KUKA KRL program: EPS_2_25694_CR03_A_20260114065856.src

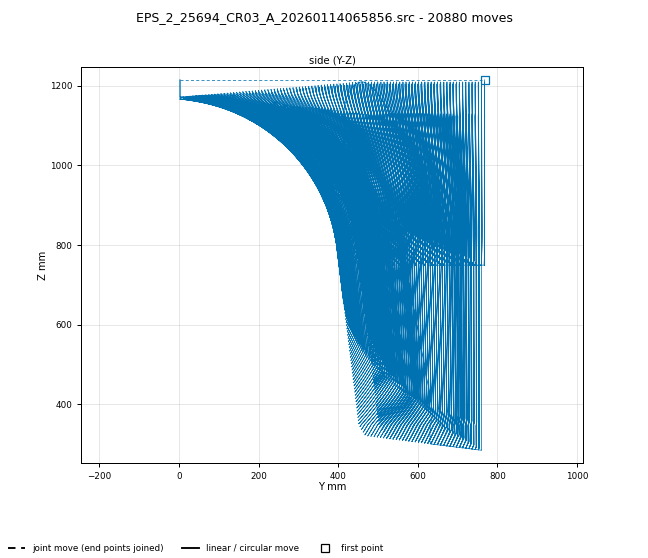
[picture p0: tool path of EPS_2_25694_CR03_A_20260114065856.src, 20880 of 20882 moves have a stored position in this frame; points joined in program order, loops and branches not executed]
&ACCESS RVP
&REL 4
&COMMENT QRS 19112012
&PARAM EDITMASK = *
DEF PART()
EXT BAS (BAS_COMMAND :IN,REAL :IN )
INT I
BAS (#INITMOV,0 )

;KUKA QRS Post kuka4.cps  Date:22-06-2017 !

File_ID=2973

QRS_PRE_INIT()

;Init var - Until changes are made in qrs_pre_init
Outlet_Square_prg=0
Inlet_1_Square_prg=0
Inlet_2_Square_prg=0
Inlet_3_Square_prg=0
Inlet_4_Square_prg=0
Inlet_5_Square_prg=0

Outlet_1={X 0.000, Y 457.000, Z 786.000, B 0.000, E1 0.000 }
Inlet_1={X 0.000, Y 514.000, Z 744.000, B 0.000, E1 189.000 }
Outlet_1_type=838
Inlet_1_type=762
;QRS#1=Sidecore dimensions
;QRS#2=825-33" Concrete
;QRS#3=750-30" Concrete
;QRS#4=
;QRS#5=
;QRS#6=
;QRS#7=
;QRS#8=
;QRS#9=S306-46
;QRS#10=S306-42L
;QRS#11=
;QRS#12=
;QRS#13=
;QRS#14=
;QRS#15=
;QRS#16=1524x152x1676 5,5'
;QRS#17=EPS Height
;QRS#18=1205
;QRS#19=*
;QRS#20= UPDATED VERSION 22-06-2017
;QRS#21=*
Outlet_Square=0650
Inlet_1_Square=0550
Inlet_2_Square=0
Inlet_3_Square=0
Inlet_4_Square=0
Inlet_5_Square=0
Mill_Square=1
Outlet_Square_Prg=267
Inlet_1_Square_prg=266

QRS_INIT()

$ADVANCE=5

; T1
PTP {E1 173.009,E2 173.009}
PTP {X 0,Y 767.725,A -85,B 0,C 180,E1 173.009,E2 173.009,E3 0,E4 0,E5 0,E6 0}
QRS_SPEED_INIT()
LIN {X 0,Y 767.725,Z 1215,A -85,B 0,C 180,E1 173.009,E2 173.009,E3 0,E4 0,E5 0,E6 0} C_VEL
LIN {X 0,Y 767.725,Z 751.56,A -85,B 0,C 180,E1 173.009,E2 173.009} C_VEL
LIN {X 0,Y 767.762,Z 749.56,A -85,B 0,C 180,E1 173.158,E2 173.158} C_VEL
LIN {X 0,Y 767.852,Z 749.56,A -85,B 0,C 180,E1 173.458,E2 173.458} C_VEL
LIN {X 0,Y 767.871,Z 749.56,A -85,B 0,C 180,E1 177.201,E2 177.201} C_VEL
LIN {X 0,Y 767.875,Z 749.56,A -85,B 0,C 180,E1 180.933,E2 180.933} C_VEL
LIN {X 0,Y 767.854,Z 749.56,A -85,B 0,C 180,E1 184.668,E2 184.668} C_VEL
LIN {X 0,Y 767.837,Z 749.56,A -85,B 0,C 180,E1 188.423,E2 188.423} C_VEL
LIN {X 0,Y 767.811,Z 749.56,A -85,B 0,C 180,E1 192.216,E2 192.216} C_VEL
LIN {X 0,Y 767.861,Z 749.56,A -85,B 0,C 180,E1 196.219,E2 196.219} C_VEL
LIN {X 0,Y 767.815,Z 749.56,A -85,B 0,C 180,E1 199.987,E2 199.987} C_VEL
LIN {X 0,Y 767.797,Z 749.56,A -85,B 0,C 180,E1 204.011,E2 204.011} C_VEL
LIN {X 0,Y 767.777,Z 749.56,A -85,B 0,C 180,E1 208.166,E2 208.166} C_VEL
LIN {X 0,Y 767.322,Z 749.56,A -85,B 0,C 180,E1 210.327,E2 210.327} C_VEL
LIN {X 0,Y 767.741,Z 749.56,A -85,B 0,C 180,E1 212.491,E2 212.491} C_VEL
LIN {X 0,Y 767.429,Z 749.56,A -85,B 0,C 180,E1 213.853,E2 213.853} C_VEL
LIN {X 0,Y 767.751,Z 749.56,A -85,B 0,C 180,E1 217.101,E2 217.101} C_VEL
LIN {X 0,Y 767.178,Z 749.56,A -85,B 0,C 180,E1 220.041,E2 220.041} C_VEL
LIN {X 0,Y 767.652,Z 749.56,A -85,B 0,C 180,E1 221.872,E2 221.872} C_VEL
LIN {X 0,Y 767.68,Z 749.56,A -85,B 0,C 180,E1 222.901,E2 222.901} C_VEL
LIN {X 0,Y 767.683,Z 749.56,A -85,B 0,C 180,E1 224.427,E2 224.427} C_VEL
LIN {X 0,Y 767.65,Z 749.56,A -85,B 0,C 180,E1 225.573,E2 225.573} C_VEL
LIN {X 0,Y 767.7,Z 749.56,A -85,B 0,C 180,E1 229.915,E2 229.915} C_VEL
LIN {X 0,Y 767.764,Z 749.56,A -85,B 0,C 180,E1 230.596,E2 230.596} C_VEL
LIN {X 0,Y 767.72,Z 749.56,A -85,B 0,C 180,E1 232.967,E2 232.967} C_VEL
LIN {X 0,Y 767.714,Z 749.56,A -85,B 0,C 180,E1 233.556,E2 233.556} C_VEL
LIN {X 0,Y 766.586,Z 750.428,A -85,B 0,C 180,E1 233.715,E2 233.715} C_VEL
LIN {X 0,Y 767.117,Z 773.995,A -85,B 0,C 180,E1 234.011,E2 234.011} C_VEL
LIN {X 0,Y 767.163,Z 809.122,A -85,B 0,C 180,E1 234.411,E2 234.411} C_VEL
LIN {X 0,Y 767.457,Z 829.921,A -85,B 0,C 180,E1 234.684,E2 234.684} C_VEL
LIN {X 0,Y 767.407,Z 846.164,A -85,B 0,C 180,E1 234.938,E2 234.938} C_VEL
LIN {X 0,Y 767.21,Z 858.585,A -85,B 0,C 180,E1 235.165,E2 235.165} C_VEL
LIN {X 0,Y 767.328,Z 875.217,A -85,B 0,C 180,E1 235.536,E2 235.536} C_VEL
LIN {X 0,Y 767.282,Z 887.767,A -85,B 0,C 180,E1 235.85,E2 235.85} C_VEL
LIN {X 0,Y 767.451,Z 900.804,A -85,B 0,C 180,E1 236.23,E2 236.23} C_VEL
LIN {X 0,Y 767.479,Z 917.969,A -85,B 0,C 180,E1 236.766,E2 236.766} C_VEL
LIN {X 0,Y 767.395,Z 931.208,A -85,B 0,C 180,E1 237.225,E2 237.225} C_VEL
LIN {X 0,Y 767.51,Z 940.173,A -85,B 0,C 180,E1 237.569,E2 237.569} C_VEL
LIN {X 0,Y 767.582,Z 955.64,A -85,B 0,C 180,E1 238.192,E2 238.192} C_VEL
LIN {X 0,Y 767.448,Z 974.022,A -85,B 0,C 180,E1 239.005,E2 239.005} C_VEL
LIN {X 0,Y 767.587,Z 991.208,A -85,B 0,C 180,E1 239.856,E2 239.856} C_VEL
LIN {X 0,Y 767.619,Z 1008.156,A -85,B 0,C 180,E1 240.771,E2 240.771} C_VEL
LIN {X 0,Y 767.612,Z 1024.962,A -85,B 0,C 180,E1 241.762,E2 241.762} C_VEL
LIN {X 0,Y 767.627,Z 1040.383,A -85,B 0,C 180,E1 242.751,E2 242.751} C_VEL
LIN {X 0,Y 767.65,Z 1055.737,A -85,B 0,C 180,E1 243.819,E2 243.819} C_VEL
LIN {X 0,Y 767.579,Z 1070.87,A -85,B 0,C 180,E1 244.96,E2 244.96} C_VEL
LIN {X 0,Y 767.603,Z 1083.468,A -85,B 0,C 180,E1 245.983,E2 245.983} C_VEL
LIN {X 0,Y 767.694,Z 1096.523,A -85,B 0,C 180,E1 247.13,E2 247.13} C_VEL
LIN {X 0,Y 767.584,Z 1109.748,A -85,B 0,C 180,E1 248.384,E2 248.384} C_VEL
LIN {X 0,Y 767.747,Z 1122.086,A -85,B 0,C 180,E1 249.663,E2 249.663} C_VEL
LIN {X 0,Y 767.589,Z 1133.958,A -85,B 0,C 180,E1 250.998,E2 250.998} C_VEL
LIN {X 0,Y 767.631,Z 1143.982,A -85,B 0,C 180,E1 252.227,E2 252.227} C_VEL
LIN {X 0,Y 767.795,Z 1151.236,A -85,B 0,C 180,E1 253.208,E2 253.208} C_VEL
LIN {X 0,Y 767.611,Z 1156.399,A -85,B 0,C 180,E1 253.933,E2 253.933} C_VEL
LIN {X 0,Y 767.552,Z 1164.121,A -85,B 0,C 180,E1 255.094,E2 255.094} C_VEL
LIN {X 0,Y 767.84,Z 1172.641,A -85,B 0,C 180,E1 256.534,E2 256.534} C_VEL
LIN {X 0,Y 767.501,Z 1180.531,A -85,B 0,C 180,E1 258.018,E2 258.018} C_VEL
LIN {X 0,Y 767.668,Z 1187.124,A -85,B 0,C 180,E1 259.448,E2 259.448} C_VEL
LIN {X 0,Y 767.832,Z 1190.052,A -85,B 0,C 180,E1 260.16,E2 260.16} C_VEL
LIN {X 0,Y 767.523,Z 1195.334,A -85,B 0,C 180,E1 261.574,E2 261.574} C_VEL
LIN {X 0,Y 767.558,Z 1198.326,A -85,B 0,C 180,E1 262.516,E2 262.516} C_VEL
LIN {X 0,Y 767.784,Z 1200.912,A -85,B 0,C 180,E1 263.458,E2 263.458} C_VEL
LIN {X 0,Y 767.79,Z 1201.883,A -85,B 0,C 180,E1 263.833,E2 263.833} C_VEL
LIN {X 0,Y 767.592,Z 1203.647,A -85,B 0,C 180,E1 264.582,E2 264.582} C_VEL
LIN {X 0,Y 767.51,Z 1205.161,A -85,B 0,C 180,E1 265.33,E2 265.33} C_VEL
LIN {X 0,Y 767.558,Z 1206.426,A -85,B 0,C 180,E1 266.079,E2 266.079} C_VEL
LIN {X 0,Y 767.836,Z 1207.855,A -85,B 0,C 180,E1 267.201,E2 267.201} C_VEL
LIN {X 0,Y 767.461,Z 1209.218,A -85,B 0,C 180,E1 269.067,E2 269.067} C_VEL
LIN {X 0,Y 767.845,Z 1209.143,A -85,B 0,C 180,E1 270.933,E2 270.933} C_VEL
LIN {X 0,Y 767.8,Z 1207.862,A -85,B 0,C 180,E1 272.799,E2 272.799} C_VEL
LIN {X 0,Y 767.607,Z 1206.417,A -85,B 0,C 180,E1 273.921,E2 273.921} C_VEL
LIN {X 0,Y 767.507,Z 1205.161,A -85,B 0,C 180,E1 274.67,E2 274.67} C_VEL
LIN {X 0,Y 767.55,Z 1203.654,A -85,B 0,C 180,E1 275.419,E2 275.419} C_VEL
LIN {X 0,Y 767.819,Z 1200.906,A -85,B 0,C 180,E1 276.542,E2 276.542} C_VEL
LIN {X 0,Y 767.591,Z 1198.32,A -85,B 0,C 180,E1 277.484,E2 277.484} C_VEL
LIN {X 0,Y 767.491,Z 1195.339,A -85,B 0,C 180,E1 278.427,E2 278.427} C_VEL
LIN {X 0,Y 767.749,Z 1190.065,A -85,B 0,C 180,E1 279.841,E2 279.841} C_VEL
LIN {X 0,Y 767.719,Z 1187.116,A -85,B 0,C 180,E1 280.552,E2 280.552} C_VEL
LIN {X 0,Y 767.49,Z 1179.366,A -85,B 0,C 180,E1 282.22,E2 282.22} C_VEL
LIN {X 0,Y 767.745,Z 1172.6,A -85,B 0,C 180,E1 283.477,E2 283.477} C_VEL
LIN {X 0,Y 767.714,Z 1168.739,A -85,B 0,C 180,E1 284.133,E2 284.133} C_VEL
LIN {X 0,Y 767.54,Z 1162.92,A -85,B 0,C 180,E1 285.1,E2 285.1} C_VEL
LIN {X 0,Y 767.667,Z 1153.06,A -85,B 0,C 180,E1 286.552,E2 286.552} C_VEL
LIN {X 0,Y 767.78,Z 1147.604,A -85,B 0,C 180,E1 287.28,E2 287.28} C_VEL
LIN {X 0,Y 767.63,Z 1142.008,A -85,B 0,C 180,E1 288.018,E2 288.018} C_VEL
LIN {X 0,Y 767.581,Z 1131.866,A -85,B 0,C 180,E1 289.249,E2 289.249} C_VEL
LIN {X 0,Y 767.776,Z 1119.932,A -85,B 0,C 180,E1 290.566,E2 290.566} C_VEL
LIN {X 0,Y 767.586,Z 1107.113,A -85,B 0,C 180,E1 291.872,E2 291.872} C_VEL
LIN {X 0,Y 767.665,Z 1095.112,A -85,B 0,C 180,E1 292.997,E2 292.997} C_VEL
LIN {X 0,Y 767.698,Z 1081.936,A -85,B 0,C 180,E1 294.142,E2 294.142} C_VEL
LIN {X 0,Y 767.621,Z 1067.008,A -85,B 0,C 180,E1 295.338,E2 295.338} C_VEL
LIN {X 0,Y 767.649,Z 1052.647,A -85,B 0,C 180,E1 296.4,E2 296.4} C_VEL
LIN {X 0,Y 767.608,Z 1037.372,A -85,B 0,C 180,E1 297.447,E2 297.447} C_VEL
LIN {X 0,Y 767.587,Z 1021.65,A -85,B 0,C 180,E1 298.44,E2 298.44} C_VEL
LIN {X 0,Y 767.552,Z 1006.46,A -85,B 0,C 180,E1 299.329,E2 299.329} C_VEL
LIN {X 0,Y 767.57,Z 987.927,A -85,B 0,C 180,E1 300.312,E2 300.312} C_VEL
LIN {X 0,Y 767.436,Z 969.608,A -85,B 0,C 180,E1 301.2,E2 301.2} C_VEL
LIN {X 0,Y 767.571,Z 952.397,A -85,B 0,C 180,E1 301.946,E2 301.946} C_VEL
LIN {X 0,Y 767.52,Z 932.768,A -85,B 0,C 180,E1 302.714,E2 302.714} C_VEL
LIN {X 0,Y 767.357,Z 920.45,A -85,B 0,C 180,E1 303.153,E2 303.153} C_VEL
LIN {X 0,Y 767.469,Z 911.2,A -85,B 0,C 180,E1 303.452,E2 303.452} C_VEL
LIN {X 0,Y 767.486,Z 892.926,A -85,B 0,C 180,E1 303.999,E2 303.999} C_VEL
LIN {X 0,Y 767.238,Z 876.515,A -85,B 0,C 180,E1 304.438,E2 304.438} C_VEL
LIN {X 0,Y 767.413,Z 858.616,A -85,B 0,C 180,E1 304.824,E2 304.824} C_VEL
LIN {X 0,Y 767.273,Z 841.666,A -85,B 0,C 180,E1 305.144,E2 305.144} C_VEL
LIN {X 0,Y 767.208,Z 834.362,A -85,B 0,C 180,E1 305.265,E2 305.265} C_VEL
LIN {X 0,Y 767.311,Z 816.709,A -85,B 0,C 180,E1 305.495,E2 305.495} C_VEL
LIN {X 0,Y 767.059,Z 771.903,A -85,B 0,C 180,E1 306.015,E2 306.015} C_VEL
LIN {X 0,Y 767.711,Z 749.56,A -85,B 0,C 180,E1 306.444,E2 306.444} C_VEL
LIN {X 0,Y 767.863,Z 749.56,A -85,B 0,C 180,E1 307.11,E2 307.11} C_VEL
LIN {X 0,Y 767.67,Z 749.56,A -85,B 0,C 180,E1 311.869,E2 311.869} C_VEL
LIN {X 0,Y 767.709,Z 749.56,A -85,B 0,C 180,E1 312.901,E2 312.901} C_VEL
LIN {X 0,Y 767.691,Z 749.56,A -85,B 0,C 180,E1 314.424,E2 314.424} C_VEL
LIN {X 0,Y 767.651,Z 749.56,A -85,B 0,C 180,E1 315.571,E2 315.571} C_VEL
LIN {X 0,Y 767.683,Z 749.56,A -85,B 0,C 180,E1 319.915,E2 319.915} C_VEL
LIN {X 0,Y 767.687,Z 749.56,A -85,B 0,C 180,E1 320.589,E2 320.589} C_VEL
LIN {X 0,Y 767.216,Z 749.56,A -85,B 0,C 180,E1 322.952,E2 322.952} C_VEL
LIN {X 0,Y 767.713,Z 749.56,A -85,B 0,C 180,E1 325.268,E2 325.268} C_VEL
LIN {X 0,Y 767.782,Z 749.56,A -85,B 0,C 180,E1 329.615,E2 329.615} C_VEL
LIN {X 0,Y 767.607,Z 749.56,A -85,B 0,C 180,E1 333.923,E2 333.923} C_VEL
LIN {X 0,Y 767.274,Z 749.56,A -85,B 0,C 180,E1 335.972,E2 335.972} C_VEL
LIN {X 0,Y 767.417,Z 749.56,A -85,B 0,C 180,E1 338.154,E2 338.154} C_VEL
LIN {X 0,Y 767.506,Z 749.56,A -85,B 0,C 180,E1 340.005,E2 340.005} C_VEL
LIN {X 0,Y 767.86,Z 749.56,A -85,B 0,C 180,E1 343.782,E2 343.782} C_VEL
LIN {X 0,Y 767.812,Z 749.56,A -85,B 0,C 180,E1 347.784,E2 347.784} C_VEL
LIN {X 0,Y 767.842,Z 749.56,A -85,B 0,C 180,E1 351.577,E2 351.577} C_VEL
LIN {X 0,Y 767.86,Z 749.56,A -85,B 0,C 180,E1 355.332,E2 355.332} C_VEL
LIN {X 0,Y 767.86,Z 749.56,A -85,B 0,C 180,E1 359.067,E2 359.067} C_VEL
LIN {X 0,Y 767.865,Z 749.56,A -85,B 0,C 180,E1 362.799,E2 362.799} C_VEL
LIN {X 0,Y 767.863,Z 749.56,A -85,B 0,C 180,E1 366.542,E2 366.542} C_VEL
LIN {X 0,Y 767.821,Z 749.56,A -85,B 0,C 180,E1 370.314,E2 370.314} C_VEL
LIN {X 0,Y 767.653,Z 749.56,A -85,B 0,C 180,E1 374.134,E2 374.134} C_VEL
LIN {X 0,Y 767.196,Z 749.56,A -85,B 0,C 180,E1 376.076,E2 376.076} C_VEL
LIN {X 0,Y 767.775,Z 749.56,A -85,B 0,C 180,E1 379.988,E2 379.988} C_VEL
LIN {X 0,Y 767.087,Z 749.56,A -85,B 0,C 180,E1 382.006,E2 382.006} C_VEL
LIN {X 0,Y 767.153,Z 749.56,A -85,B 0,C 180,E1 384.033,E2 384.033} C_VEL
LIN {X 0,Y 767.608,Z 749.56,A -85,B 0,C 180,E1 386.077,E2 386.077} C_VEL
LIN {X 0,Y 767.763,Z 749.56,A -85,B 0,C 180,E1 390.383,E2 390.383} C_VEL
LIN {X 0,Y 767.703,Z 749.56,A -85,B 0,C 180,E1 394.733,E2 394.733} C_VEL
LIN {X 0,Y 767.231,Z 749.56,A -85,B 0,C 180,E1 397.062,E2 397.062} C_VEL
LIN {X 0,Y 767.703,Z 749.56,A -85,B 0,C 180,E1 399.41,E2 399.41} C_VEL
LIN {X 0,Y 767.697,Z 749.56,A -85,B 0,C 180,E1 400.087,E2 400.087} C_VEL
LIN {X 0,Y 767.632,Z 749.56,A -85,B 0,C 180,E1 404.43,E2 404.43} C_VEL
LIN {X 0,Y 767.623,Z 749.56,A -85,B 0,C 180,E1 405.571,E2 405.571} C_VEL
LIN {X 0,Y 767.8,Z 749.56,A -85,B 0,C 180,E1 408.14,E2 408.14} C_VEL
LIN {X 0,Y 767.744,Z 749.56,A -85,B 0,C 180,E1 408.467,E2 408.467} C_VEL
LIN {X 0,Y 767.495,Z 749.56,A -85,B 0,C 180,E1 408.516,E2 408.516} C_VEL
LIN {X 0,Y 766.821,Z 752.052,A -85,B 0,C 180,E1 408.631,E2 408.631} C_VEL
LIN {X 0,Y 767.435,Z 777.541,A -85,B 0,C 180,E1 408.952,E2 408.952} C_VEL
LIN {X 0,Y 767.536,Z 790.523,A -85,B 0,C 180,E1 409.135,E2 409.135} C_VEL
LIN {X 0,Y 767.35,Z 808.543,A -85,B 0,C 180,E1 409.442,E2 409.442} C_VEL
LIN {X 0,Y 767.534,Z 826.704,A -85,B 0,C 180,E1 409.843,E2 409.843} C_VEL
LIN {X 0,Y 767.439,Z 844.838,A -85,B 0,C 180,E1 410.306,E2 410.306} C_VEL
LIN {X 0,Y 767.613,Z 862.804,A -85,B 0,C 180,E1 410.854,E2 410.854} C_VEL
LIN {X 0,Y 767.622,Z 879.893,A -85,B 0,C 180,E1 411.44,E2 411.44} C_VEL
LIN {X 0,Y 767.529,Z 896,A -85,B 0,C 180,E1 412.056,E2 412.056} C_VEL
LIN {X 0,Y 767.641,Z 913.554,A -85,B 0,C 180,E1 412.818,E2 412.818} C_VEL
LIN {X 0,Y 767.603,Z 930.122,A -85,B 0,C 180,E1 413.61,E2 413.61} C_VEL
LIN {X 0,Y 767.646,Z 945.53,A -85,B 0,C 180,E1 414.423,E2 414.423} C_VEL
LIN {X 0,Y 767.659,Z 960.2,A -85,B 0,C 180,E1 415.266,E2 415.266} C_VEL
LIN {X 0,Y 767.657,Z 975.595,A -85,B 0,C 180,E1 416.235,E2 416.235} C_VEL
LIN {X 0,Y 767.656,Z 988.606,A -85,B 0,C 180,E1 417.121,E2 417.121} C_VEL
LIN {X 0,Y 767.705,Z 1003.063,A -85,B 0,C 180,E1 418.197,E2 418.197} C_VEL
LIN {X 0,Y 767.703,Z 1014.97,A -85,B 0,C 180,E1 419.152,E2 419.152} C_VEL
LIN {X 0,Y 767.62,Z 1027.03,A -85,B 0,C 180,E1 420.197,E2 420.197} C_VEL
LIN {X 0,Y 767.738,Z 1038.105,A -85,B 0,C 180,E1 421.238,E2 421.238} C_VEL
LIN {X 0,Y 767.706,Z 1046.555,A -85,B 0,C 180,E1 422.096,E2 422.096} C_VEL
LIN {X 0,Y 767.604,Z 1052.669,A -85,B 0,C 180,E1 422.75,E2 422.75} C_VEL
LIN {X 0,Y 767.607,Z 1059.972,A -85,B 0,C 180,E1 423.564,E2 423.564} C_VEL
LIN {X 0,Y 767.83,Z 1069.922,A -85,B 0,C 180,E1 424.785,E2 424.785} C_VEL
LIN {X 0,Y 767.567,Z 1078.916,A -85,B 0,C 180,E1 425.982,E2 425.982} C_VEL
LIN {X 0,Y 767.62,Z 1087.471,A -85,B 0,C 180,E1 427.254,E2 427.254} C_VEL
LIN {X 0,Y 767.83,Z 1093.635,A -85,B 0,C 180,E1 428.284,E2 428.284} C_VEL
LIN {X 0,Y 767.666,Z 1097.591,A -85,B 0,C 180,E1 428.983,E2 428.983} C_VEL
LIN {X 0,Y 767.59,Z 1103.012,A -85,B 0,C 180,E1 430.008,E2 430.008} C_VEL
LIN {X 0,Y 767.812,Z 1108.759,A -85,B 0,C 180,E1 431.25,E2 431.25} C_VEL
LIN {X 0,Y 767.548,Z 1113.714,A -85,B 0,C 180,E1 432.47,E2 432.47} C_VEL
LIN {X 0,Y 767.56,Z 1118.734,A -85,B 0,C 180,E1 433.932,E2 433.932} C_VEL
LIN {X 0,Y 767.778,Z 1121.922,A -85,B 0,C 180,E1 435.098,E2 435.098} C_VEL
LIN {X 0,Y 767.555,Z 1124.663,A -85,B 0,C 180,E1 436.287,E2 436.287} C_VEL
LIN {X 0,Y 767.561,Z 1125.789,A -85,B 0,C 180,E1 436.825,E2 436.825} C_VEL
LIN {X 0,Y 767.726,Z 1127.188,A -85,B 0,C 180,E1 437.783,E2 437.783} C_VEL
LIN {X 0,Y 767.687,Z 1128.292,A -85,B 0,C 180,E1 438.735,E2 438.735} C_VEL
LIN {X 0,Y 767.547,Z 1129.111,A -85,B 0,C 180,E1 439.683,E2 439.683} C_VEL
LIN {X 0,Y 767.826,Z 1129.242,A -85,B 0,C 180,E1 441.577,E2 441.577} C_VEL
LIN {X 0,Y 767.83,Z 1128.015,A -85,B 0,C 180,E1 443.458,E2 443.458} C_VEL
LIN {X 0,Y 767.589,Z 1126.531,A -85,B 0,C 180,E1 444.582,E2 444.582} C_VEL
LIN {X 0,Y 767.564,Z 1125.284,A -85,B 0,C 180,E1 445.331,E2 445.331} C_VEL
LIN {X 0,Y 767.679,Z 1123.677,A -85,B 0,C 180,E1 446.08,E2 446.08} C_VEL
LIN {X 0,Y 767.798,Z 1121.875,A -85,B 0,C 180,E1 446.828,E2 446.828} C_VEL
LIN {X 0,Y 767.544,Z 1118.842,A -85,B 0,C 180,E1 447.947,E2 447.947} C_VEL
LIN {X 0,Y 767.622,Z 1113.698,A -85,B 0,C 180,E1 449.44,E2 449.44} C_VEL
LIN {X 0,Y 767.831,Z 1110.655,A -85,B 0,C 180,E1 450.186,E2 450.186} C_VEL
LIN {X 0,Y 767.664,Z 1107.52,A -85,B 0,C 180,E1 450.933,E2 450.933} C_VEL
LIN {X 0,Y 767.556,Z 1102.294,A -85,B 0,C 180,E1 452.053,E2 452.053} C_VEL
LIN {X 0,Y 767.799,Z 1095.255,A -85,B 0,C 180,E1 453.359,E2 453.359} C_VEL
LIN {X 0,Y 767.573,Z 1087.396,A -85,B 0,C 180,E1 454.669,E2 454.669} C_VEL
LIN {X 0,Y 767.62,Z 1078.527,A -85,B 0,C 180,E1 455.98,E2 455.98} C_VEL
LIN {X 0,Y 767.792,Z 1071.247,A -85,B 0,C 180,E1 456.948,E2 456.948} C_VEL
LIN {X 0,Y 767.675,Z 1067.061,A -85,B 0,C 180,E1 457.483,E2 457.483} C_VEL
LIN {X 0,Y 767.588,Z 1058.245,A -85,B 0,C 180,E1 458.543,E2 458.543} C_VEL
LIN {X 0,Y 767.766,Z 1047.447,A -85,B 0,C 180,E1 459.722,E2 459.722} C_VEL
LIN {X 0,Y 767.634,Z 1036.904,A -85,B 0,C 180,E1 460.79,E2 460.79} C_VEL
LIN {X 0,Y 767.598,Z 1024.027,A -85,B 0,C 180,E1 461.98,E2 461.98} C_VEL
LIN {X 0,Y 767.723,Z 1012.854,A -85,B 0,C 180,E1 462.933,E2 462.933} C_VEL
LIN {X 0,Y 767.665,Z 1000.11,A -85,B 0,C 180,E1 463.943,E2 463.943} C_VEL
LIN {X 0,Y 767.679,Z 986.955,A -85,B 0,C 180,E1 464.904,E2 464.904} C_VEL
LIN {X 0,Y 767.69,Z 972.569,A -85,B 0,C 180,E1 465.871,E2 465.871} C_VEL
LIN {X 0,Y 767.661,Z 957.622,A -85,B 0,C 180,E1 466.795,E2 466.795} C_VEL
LIN {X 0,Y 767.63,Z 942.545,A -85,B 0,C 180,E1 467.65,E2 467.65} C_VEL
LIN {X 0,Y 767.662,Z 927.156,A -85,B 0,C 180,E1 468.447,E2 468.447} C_VEL
LIN {X 0,Y 767.629,Z 910.076,A -85,B 0,C 180,E1 469.248,E2 469.248} C_VEL
LIN {X 0,Y 767.544,Z 895.631,A -85,B 0,C 180,E1 469.869,E2 469.869} C_VEL
LIN {X 0,Y 767.649,Z 876.582,A -85,B 0,C 180,E1 470.588,E2 470.588} C_VEL
LIN {X 0,Y 767.536,Z 859.243,A -85,B 0,C 180,E1 471.174,E2 471.174} C_VEL
LIN {X 0,Y 767.439,Z 851.693,A -85,B 0,C 180,E1 471.401,E2 471.401} C_VEL
LIN {X 0,Y 767.597,Z 839.263,A -85,B 0,C 180,E1 471.747,E2 471.747} C_VEL
LIN {X 0,Y 767.593,Z 822.318,A -85,B 0,C 180,E1 472.166,E2 472.166} C_VEL
LIN {X 0,Y 767.358,Z 804.891,A -85,B 0,C 180,E1 472.539,E2 472.539} C_VEL
LIN {X 0,Y 767.603,Z 785.386,A -85,B 0,C 180,E1 472.849,E2 472.849} C_VEL
LIN {X 0,Y 767.457,Z 763.559,A -85,B 0,C 180,E1 473.125,E2 473.125} C_VEL
LIN {X 0,Y 767.242,Z 750.234,A -85,B 0,C 180,E1 473.279,E2 473.279} C_VEL
LIN {X 0,Y 767.612,Z 749.56,A -85,B 0,C 180,E1 473.402,E2 473.402} C_VEL
LIN {X 0,Y 767.779,Z 749.56,A -85,B 0,C 180,E1 473.519,E2 473.519} C_VEL
LIN {X 0,Y 767.721,Z 749.56,A -85,B 0,C 180,E1 474.013,E2 474.013} C_VEL
LIN {X 0,Y 767.754,Z 749.56,A -85,B 0,C 180,E1 478.166,E2 478.166} C_VEL
LIN {X 0,Y 767.295,Z 749.56,A -85,B 0,C 180,E1 480.324,E2 480.324} C_VEL
LIN {X 0,Y 767.681,Z 749.56,A -85,B 0,C 180,E1 482.492,E2 482.492} C_VEL
LIN {X 0,Y 767.38,Z 749.56,A -85,B 0,C 180,E1 483.844,E2 483.844} C_VEL
LIN {X 0,Y 767.71,Z 749.56,A -85,B 0,C 180,E1 487.095,E2 487.095} C_VEL
LIN {X 0,Y 767.179,Z 749.56,A -85,B 0,C 180,E1 490.038,E2 490.038} C_VEL
LIN {X 0,Y 767.685,Z 749.56,A -85,B 0,C 180,E1 491.868,E2 491.868} C_VEL
LIN {X 0,Y 767.69,Z 749.56,A -85,B 0,C 180,E1 492.9,E2 492.9} C_VEL
LIN {X 0,Y 767.647,Z 749.56,A -85,B 0,C 180,E1 494.427,E2 494.427} C_VEL
LIN {X 0,Y 767.613,Z 749.56,A -85,B 0,C 180,E1 495.568,E2 495.568} C_VEL
LIN {X 0,Y 767.701,Z 749.56,A -85,B 0,C 180,E1 499.913,E2 499.913} C_VEL
LIN {X 0,Y 767.709,Z 749.56,A -85,B 0,C 180,E1 500.591,E2 500.591} C_VEL
LIN {X 0,Y 767.216,Z 749.56,A -85,B 0,C 180,E1 502.951,E2 502.951} C_VEL
LIN {X 0,Y 767.693,Z 749.56,A -85,B 0,C 180,E1 505.267,E2 505.267} C_VEL
LIN {X 0,Y 767.744,Z 749.56,A -85,B 0,C 180,E1 509.619,E2 509.619} C_VEL
LIN {X 0,Y 767.62,Z 749.56,A -85,B 0,C 180,E1 513.924,E2 513.924} C_VEL
LIN {X 0,Y 767.163,Z 749.56,A -85,B 0,C 180,E1 515.968,E2 515.968} C_VEL
LIN {X 0,Y 767.125,Z 749.56,A -85,B 0,C 180,E1 518.209,E2 518.209} C_VEL
LIN {X 0,Y 767.758,Z 749.56,A -85,B 0,C 180,E1 520.012,E2 520.012} C_VEL
LIN {X 0,Y 767.192,Z 749.56,A -85,B 0,C 180,E1 523.954,E2 523.954} C_VEL
LIN {X 0,Y 767.636,Z 749.56,A -85,B 0,C 180,E1 525.865,E2 525.865} C_VEL
LIN {X 0,Y 767.816,Z 749.56,A -85,B 0,C 180,E1 529.686,E2 529.686} C_VEL
LIN {X 0,Y 767.762,Z 749.56,A -85,B 0,C 180,E1 533.158,E2 533.158} C_VEL
LIN {X 0,Y 765.233,Z 749.56,A -85,B 0,C 180,E1 534.117,E2 534.117} C_VEL
LIN {X 0,Y 759.658,Z 749.56,A -85,B 0,C 180,E1 535.545,E2 535.545} C_VEL
LIN {X 0,Y 759.576,Z 749.56,A -85,B 0,C 180,E1 535.711,E2 535.711} C_VEL
LIN {X 0,Y 759.694,Z 749.56,A -85,B 0,C 180,E1 539.997,E2 539.997} C_VEL
LIN {X 0,Y 759.906,Z 749.56,A -85,B 0,C 180,E1 544.559,E2 544.559} C_VEL
LIN {X 0,Y 759.684,Z 749.56,A -85,B 0,C 180,E1 549.154,E2 549.154} C_VEL
LIN {X 0,Y 759.483,Z 749.56,A -85,B 0,C 180,E1 553.811,E2 553.811} C_VEL
LIN {X 0,Y 759.604,Z 749.56,A -85,B 0,C 180,E1 557.359,E2 557.359} C_VEL
LIN {X 0,Y 759.573,Z 749.56,A -85,B 0,C 180,E1 560.981,E2 560.981} C_VEL
LIN {X 0,Y 759.629,Z 749.56,A -85,B 0,C 180,E1 564.69,E2 564.69} C_VEL
LIN {X 0,Y 759.614,Z 749.56,A -85,B 0,C 180,E1 568.917,E2 568.917} C_VEL
LIN {X 0,Y 759.606,Z 749.56,A -85,B 0,C 180,E1 573.328,E2 573.328} C_VEL
LIN {X 0,Y 759.453,Z 749.56,A -85,B 0,C 180,E1 578.082,E2 578.082} C_VEL
LIN {X 0,Y 759.777,Z 749.56,A -85,B 0,C 180,E1 582.616,E2 582.616} C_VEL
LIN {X 0,Y 759.616,Z 749.56,A -85,B 0,C 180,E1 585.871,E2 585.871} C_VEL
LIN {X 0,Y 759.814,Z 749.56,A -85,B 0,C 180,E1 590.86,E2 590.86} C_VEL
LIN {X 0,Y 759.812,Z 749.589,A -85,B 0,C 180,E1 593.329,E2 593.329} C_VEL
LIN {X 0,Y 760.891,Z 847.417,A -85,B 0,C 180,E1 594.616,E2 594.616} C_VEL
LIN {X 0,Y 760.732,Z 894.139,A -85,B 0,C 180,E1 595.691,E2 595.691} C_VEL
LIN {X 0,Y 760.628,Z 940.818,A -85,B 0,C 180,E1 597.264,E2 597.264} C_VEL
LIN {X 0,Y 760.469,Z 986.538,A -85,B 0,C 180,E1 599.306,E2 599.306} C_VEL
LIN {X 0,Y 760.302,Z 1028.129,A -85,B 0,C 180,E1 601.671,E2 601.671} C_VEL
LIN {X 0,Y 760.108,Z 1068.911,A -85,B 0,C 180,E1 604.537,E2 604.537} C_VEL
LIN {X 0,Y 759.935,Z 1106.116,A -85,B 0,C 180,E1 607.801,E2 607.801} C_VEL
LIN {X 0,Y 759.817,Z 1135.562,A -85,B 0,C 180,E1 610.993,E2 610.993} C_VEL
LIN {X 0,Y 759.749,Z 1158.904,A -85,B 0,C 180,E1 614.128,E2 614.128} C_VEL
LIN {X 0,Y 759.745,Z 1178,A -85,B 0,C 180,E1 617.361,E2 617.361} C_VEL
LIN {X 0,Y 759.772,Z 1193.413,A -85,B 0,C 180,E1 620.844,E2 620.844} C_VEL
LIN {X 0,Y 759.773,Z 1203.568,A -85,B 0,C 180,E1 624.292,E2 624.292} C_VEL
LIN {X 0,Y 759.787,Z 1208.98,A -85,B 0,C 180,E1 627.72,E2 627.72} C_VEL
LIN {X 0,Y 759.929,Z 1209.669,A -85,B 0,C 180,E1 631.139,E2 631.139} C_VEL
LIN {X 0,Y 759.659,Z 1205.912,A -85,B 0,C 180,E1 634.563,E2 634.563} C_VEL
LIN {X 0,Y 759.648,Z 1197.335,A -85,B 0,C 180,E1 638.004,E2 638.004} C_VEL
LIN {X 0,Y 759.701,Z 1185.042,A -85,B 0,C 180,E1 641.182,E2 641.182} C_VEL
LIN {X 0,Y 759.769,Z 1166.458,A -85,B 0,C 180,E1 644.689,E2 644.689} C_VEL
LIN {X 0,Y 759.851,Z 1142.884,A -85,B 0,C 180,E1 648.103,E2 648.103} C_VEL
LIN {X 0,Y 759.941,Z 1112.255,A -85,B 0,C 180,E1 651.584,E2 651.584} C_VEL
LIN {X 0,Y 760.107,Z 1078.537,A -85,B 0,C 180,E1 654.676,E2 654.676} C_VEL
LIN {X 0,Y 760.272,Z 1039.395,A -85,B 0,C 180,E1 657.604,E2 657.604} C_VEL
LIN {X 0,Y 760.418,Z 995.971,A -85,B 0,C 180,E1 660.199,E2 660.199} C_VEL
LIN {X 0,Y 760.66,Z 954.474,A -85,B 0,C 180,E1 662.184,E2 662.184} C_VEL
LIN {X 0,Y 760.762,Z 909.659,A -85,B 0,C 180,E1 663.834,E2 663.834} C_VEL
LIN {X 0,Y 760.853,Z 864.887,A -85,B 0,C 180,E1 665.036,E2 665.036} C_VEL
LIN {X 0,Y 760.878,Z 820.374,A -85,B 0,C 180,E1 665.795,E2 665.795} C_VEL
LIN {X 0,Y 759.855,Z 749.643,A -85,B 0,C 180,E1 666.668,E2 666.668} C_VEL
LIN {X 0,Y 759.774,Z 749.56,A -85,B 0,C 180,E1 672.62,E2 672.62} C_VEL
LIN {X 0,Y 759.621,Z 749.56,A -85,B 0,C 180,E1 675.875,E2 675.875} C_VEL
LIN {X 0,Y 759.686,Z 749.56,A -85,B 0,C 180,E1 680.874,E2 680.874} C_VEL
LIN {X 0,Y 759.482,Z 749.56,A -85,B 0,C 180,E1 686.147,E2 686.147} C_VEL
LIN {X 0,Y 759.632,Z 749.56,A -85,B 0,C 180,E1 690.18,E2 690.18} C_VEL
LIN {X 0,Y 759.377,Z 749.56,A -85,B 0,C 180,E1 695.301,E2 695.301} C_VEL
LIN {X 0,Y 759.54,Z 749.56,A -85,B 0,C 180,E1 700.234,E2 700.234} C_VEL
LIN {X 0,Y 759.942,Z 749.56,A -85,B 0,C 180,E1 703.839,E2 703.839} C_VEL
LIN {X 0,Y 759.655,Z 749.56,A -85,B 0,C 180,E1 708.529,E2 708.529} C_VEL
LIN {X 0,Y 759.571,Z 749.56,A -85,B 0,C 180,E1 713.147,E2 713.147} C_VEL
LIN {X 0,Y 759.602,Z 749.56,A -85,B 0,C 180,E1 716.582,E2 716.582} C_VEL
LIN {X 0,Y 759.661,Z 749.56,A -85,B 0,C 180,E1 720.003,E2 720.003} C_VEL
LIN {X 0,Y 759.574,Z 749.56,A -85,B 0,C 180,E1 724.568,E2 724.568} C_VEL
LIN {X 0,Y 759.567,Z 749.56,A -85,B 0,C 180,E1 728.009,E2 728.009} C_VEL
LIN {X 0,Y 759.512,Z 749.56,A -85,B 0,C 180,E1 731.48,E2 731.48} C_VEL
LIN {X 0,Y 759.458,Z 749.56,A -85,B 0,C 180,E1 734.995,E2 734.995} C_VEL
LIN {X 0,Y 759.518,Z 749.56,A -85,B 0,C 180,E1 740.756,E2 740.756} C_VEL
LIN {X 0,Y 759.545,Z 749.56,A -85,B 0,C 180,E1 746.457,E2 746.457} C_VEL
LIN {X 0,Y 759.53,Z 749.56,A -85,B 0,C 180,E1 751.185,E2 751.185} C_VEL
LIN {X 0,Y 759.565,Z 749.56,A -85,B 0,C 180,E1 755.346,E2 755.346} C_VEL
LIN {X 0,Y 759.82,Z 749.56,A -85,B 0,C 180,E1 759.53,E2 759.53} C_VEL
LIN {X 0,Y 759.708,Z 749.56,A -85,B 0,C 180,E1 765.737,E2 765.737} C_VEL
LIN {X 0,Y 759.887,Z 749.56,A -85,B 0,C 180,E1 768.259,E2 768.259} C_VEL
LIN {X 0,Y 760.608,Z 808.436,A -85,B 0,C 180,E1 769.128,E2 769.128} C_VEL
LIN {X 0,Y 760.629,Z 856.213,A -85,B 0,C 180,E1 770.341,E2 770.341} C_VEL
LIN {X 0,Y 760.417,Z 899.885,A -85,B 0,C 180,E1 771.928,E2 771.928} C_VEL
LIN {X 0,Y 760.343,Z 944.372,A -85,B 0,C 180,E1 774.081,E2 774.081} C_VEL
LIN {X 0,Y 760.173,Z 986.556,A -85,B 0,C 180,E1 776.727,E2 776.727} C_VEL
LIN {X 0,Y 759.99,Z 1022.018,A -85,B 0,C 180,E1 779.534,E2 779.534} C_VEL
LIN {X 0,Y 759.898,Z 1051.812,A -85,B 0,C 180,E1 782.462,E2 782.462} C_VEL
LIN {X 0,Y 759.795,Z 1077.001,A -85,B 0,C 180,E1 785.556,E2 785.556} C_VEL
LIN {X 0,Y 759.875,Z 1097.413,A -85,B 0,C 180,E1 788.784,E2 788.784} C_VEL
LIN {X 0,Y 759.742,Z 1112.692,A -85,B 0,C 180,E1 792.044,E2 792.044} C_VEL
LIN {X 0,Y 759.787,Z 1123.797,A -85,B 0,C 180,E1 795.605,E2 795.605} C_VEL
LIN {X 0,Y 759.807,Z 1128.669,A -85,B 0,C 180,E1 798.529,E2 798.529} C_VEL
LIN {X 0,Y 759.909,Z 1129.698,A -85,B 0,C 180,E1 801.999,E2 801.999} C_VEL
LIN {X 0,Y 759.707,Z 1125.623,A -85,B 0,C 180,E1 805.437,E2 805.437} C_VEL
LIN {X 0,Y 759.653,Z 1118.315,A -85,B 0,C 180,E1 808.291,E2 808.291} C_VEL
LIN {X 0,Y 759.719,Z 1106.01,A -85,B 0,C 180,E1 811.425,E2 811.425} C_VEL
LIN {X 0,Y 759.737,Z 1089.033,A -85,B 0,C 180,E1 814.564,E2 814.564} C_VEL
LIN {X 0,Y 759.846,Z 1065.453,A -85,B 0,C 180,E1 817.859,E2 817.859} C_VEL
LIN {X 0,Y 759.933,Z 1038.038,A -85,B 0,C 180,E1 820.89,E2 820.89} C_VEL
LIN {X 0,Y 760.09,Z 1003.118,A -85,B 0,C 180,E1 823.949,E2 823.949} C_VEL
LIN {X 0,Y 760.261,Z 965.095,A -85,B 0,C 180,E1 826.603,E2 826.603} C_VEL
LIN {X 0,Y 760.448,Z 924.86,A -85,B 0,C 180,E1 828.84,E2 828.84} C_VEL
LIN {X 0,Y 760.619,Z 881.71,A -85,B 0,C 180,E1 830.698,E2 830.698} C_VEL
LIN {X 0,Y 760.754,Z 839.567,A -85,B 0,C 180,E1 832.047,E2 832.047} C_VEL
LIN {X 0,Y 760.774,Z 794.627,A -85,B 0,C 180,E1 833.021,E2 833.021} C_VEL
LIN {X 0,Y 759.877,Z 749.56,A -85,B 0,C 180,E1 833.643,E2 833.643} C_VEL
LIN {X 0,Y 759.597,Z 749.56,A -85,B 0,C 180,E1 838.907,E2 838.907} C_VEL
LIN {X 0,Y 759.564,Z 749.56,A -85,B 0,C 180,E1 843.316,E2 843.316} C_VEL
LIN {X 0,Y 759.432,Z 749.56,A -85,B 0,C 180,E1 848.087,E2 848.087} C_VEL
LIN {X 0,Y 759.795,Z 749.56,A -85,B 0,C 180,E1 852.612,E2 852.612} C_VEL
LIN {X 0,Y 759.586,Z 749.56,A -85,B 0,C 180,E1 855.864,E2 855.864} C_VEL
LIN {X 0,Y 759.707,Z 749.56,A -85,B 0,C 180,E1 860.874,E2 860.874} C_VEL
LIN {X 0,Y 759.448,Z 749.56,A -85,B 0,C 180,E1 866.137,E2 866.137} C_VEL
LIN {X 0,Y 759.607,Z 749.56,A -85,B 0,C 180,E1 870.171,E2 870.171} C_VEL
LIN {X 0,Y 759.689,Z 749.56,A -85,B 0,C 180,E1 874.044,E2 874.044} C_VEL
LIN {X 0,Y 759.724,Z 749.56,A -85,B 0,C 180,E1 880.233,E2 880.233} C_VEL
LIN {X 0,Y 759.619,Z 749.56,A -85,B 0,C 180,E1 886.185,E2 886.185} C_VEL
LIN {X 0,Y 759.936,Z 749.56,A -85,B 0,C 180,E1 889.687,E2 889.687} C_VEL
LIN {X 0,Y 759.695,Z 749.56,A -85,B 0,C 180,E1 894.289,E2 894.289} C_VEL
LIN {X 0,Y 759.576,Z 749.56,A -85,B 0,C 180,E1 895.711,E2 895.711} C_VEL
LIN {X 0,Y 755.755,Z 749.56,A -85,B 0,C 180,E1 896.999,E2 896.999} C_VEL
LIN {X 0,Y 751.733,Z 749.56,A -85,B 0,C 180,E1 898.301,E2 898.301} C_VEL
LIN {X 0,Y 751.712,Z 749.56,A -85,B 0,C 180,E1 902.301,E2 902.301} C_VEL
LIN {X 0,Y 751.741,Z 749.56,A -85,B 0,C 180,E1 905.765,E2 905.765} C_VEL
LIN {X 0,Y 751.641,Z 749.56,A -85,B 0,C 180,E1 909.895,E2 909.895} C_VEL
LIN {X 0,Y 751.578,Z 749.56,A -85,B 0,C 180,E1 913.959,E2 913.959} C_VEL
LIN {X 0,Y 751.675,Z 749.56,A -85,B 0,C 180,E1 917.548,E2 917.548} C_VEL
LIN {X 0,Y 751.626,Z 749.56,A -85,B 0,C 180,E1 921.213,E2 921.213} C_VEL
LIN {X 0,Y 751.625,Z 749.56,A -85,B 0,C 180,E1 925.214,E2 925.214} C_VEL
LIN {X 0,Y 751.735,Z 749.56,A -85,B 0,C 180,E1 928.842,E2 928.842} C_VEL
LIN {X 0,Y 751.844,Z 749.56,A -85,B 0,C 180,E1 932.863,E2 932.863} C_VEL
LIN {X 0,Y 751.822,Z 749.56,A -85,B 0,C 180,E1 937.081,E2 937.081} C_VEL
LIN {X 0,Y 751.822,Z 749.56,A -85,B 0,C 180,E1 943.106,E2 943.106} C_VEL
LIN {X 0,Y 751.407,Z 749.56,A -85,B 0,C 180,E1 946.861,E2 946.861} C_VEL
LIN {X 0,Y 751.829,Z 749.56,A -85,B 0,C 180,E1 951.613,E2 951.613} C_VEL
LIN {X 0,Y 751.899,Z 749.722,A -85,B 0,C 180,E1 952.88,E2 952.88} C_VEL
LIN {X 0,Y 754.01,Z 757.934,A -85,B 0,C 180,E1 953.098,E2 953.098} C_VEL
LIN {X 0,Y 754.454,Z 846.605,A -85,B 0,C 180,E1 954.254,E2 954.254} C_VEL
LIN {X 0,Y 754.05,Z 892.321,A -85,B 0,C 180,E1 955.293,E2 955.293} C_VEL
LIN {X 0,Y 753.812,Z 939.54,A -85,B 0,C 180,E1 956.879,E2 956.879} C_VEL
LIN {X 0,Y 753.394,Z 985.778,A -85,B 0,C 180,E1 958.949,E2 958.949} C_VEL
LIN {X 0,Y 753.055,Z 1027.456,A -85,B 0,C 180,E1 961.329,E2 961.329} C_VEL
LIN {X 0,Y 752.65,Z 1069.01,A -85,B 0,C 180,E1 964.274,E2 964.274} C_VEL
LIN {X 0,Y 752.33,Z 1106.118,A -85,B 0,C 180,E1 967.564,E2 967.564} C_VEL
LIN {X 0,Y 752.073,Z 1135.579,A -85,B 0,C 180,E1 970.792,E2 970.792} C_VEL
LIN {X 0,Y 751.93,Z 1160.758,A -85,B 0,C 180,E1 974.239,E2 974.239} C_VEL
LIN {X 0,Y 751.859,Z 1179.553,A -85,B 0,C 180,E1 977.522,E2 977.522} C_VEL
LIN {X 0,Y 751.835,Z 1194.427,A -85,B 0,C 180,E1 981.038,E2 981.038} C_VEL
LIN {X 0,Y 751.902,Z 1203.568,A -85,B 0,C 180,E1 984.232,E2 984.232} C_VEL
LIN {X 0,Y 751.887,Z 1208.977,A -85,B 0,C 180,E1 987.696,E2 987.696} C_VEL
LIN {X 0,Y 752.027,Z 1209.669,A -85,B 0,C 180,E1 991.151,E2 991.151} C_VEL
LIN {X 0,Y 751.768,Z 1205.912,A -85,B 0,C 180,E1 994.611,E2 994.611} C_VEL
LIN {X 0,Y 751.747,Z 1197.335,A -85,B 0,C 180,E1 998.088,E2 998.088} C_VEL
LIN {X 0,Y 751.819,Z 1185.043,A -85,B 0,C 180,E1 1001.301,E2 1001.301} C_VEL
LIN {X 0,Y 751.906,Z 1166.459,A -85,B 0,C 180,E1 1004.847,E2 1004.847} C_VEL
LIN {X 0,Y 752.036,Z 1142.882,A -85,B 0,C 180,E1 1008.298,E2 1008.298} C_VEL
LIN {X 0,Y 752.244,Z 1112.257,A -85,B 0,C 180,E1 1011.816,E2 1011.816} C_VEL
LIN {X 0,Y 752.571,Z 1078.537,A -85,B 0,C 180,E1 1014.939,E2 1014.939} C_VEL
LIN {X 0,Y 752.943,Z 1039.101,A -85,B 0,C 180,E1 1017.916,E2 1017.916} C_VEL
LIN {X 0,Y 753.36,Z 994.875,A -85,B 0,C 180,E1 1020.573,E2 1020.573} C_VEL
LIN {X 0,Y 753.791,Z 953.686,A -85,B 0,C 180,E1 1022.549,E2 1022.549} C_VEL
LIN {X 0,Y 754.083,Z 907.991,A -85,B 0,C 180,E1 1024.227,E2 1024.227} C_VEL
LIN {X 0,Y 754.327,Z 865.238,A -85,B 0,C 180,E1 1025.376,E2 1025.376} C_VEL
LIN {X 0,Y 754.476,Z 819.086,A -85,B 0,C 180,E1 1026.163,E2 1026.163} C_VEL
LIN {X 0,Y 753.352,Z 753.96,A -85,B 0,C 180,E1 1026.986,E2 1026.986} C_VEL
LIN {X 0,Y 751.996,Z 749.56,A -85,B 0,C 180,E1 1027.176,E2 1027.176} C_VEL
LIN {X 0,Y 751.817,Z 749.56,A -85,B 0,C 180,E1 1033.652,E2 1033.652} C_VEL
LIN {X 0,Y 751.392,Z 749.56,A -85,B 0,C 180,E1 1038.423,E2 1038.423} C_VEL
LIN {X 0,Y 751.545,Z 749.56,A -85,B 0,C 180,E1 1041.643,E2 1041.643} C_VEL
LIN {X 0,Y 751.573,Z 749.56,A -85,B 0,C 180,E1 1045.741,E2 1045.741} C_VEL
LIN {X 0,Y 751.702,Z 749.56,A -85,B 0,C 180,E1 1049.833,E2 1049.833} C_VEL
LIN {X 0,Y 751.509,Z 749.56,A -85,B 0,C 180,E1 1055.025,E2 1055.025} C_VEL
LIN {X 0,Y 751.609,Z 749.56,A -85,B 0,C 180,E1 1060.017,E2 1060.017} C_VEL
LIN {X 0,Y 751.706,Z 749.56,A -85,B 0,C 180,E1 1064.854,E2 1064.854} C_VEL
LIN {X 0,Y 751.752,Z 749.56,A -85,B 0,C 180,E1 1068.407,E2 1068.407} C_VEL
LIN {X 0,Y 751.676,Z 749.56,A -85,B 0,C 180,E1 1073.075,E2 1073.075} C_VEL
LIN {X 0,Y 751.729,Z 749.56,A -85,B 0,C 180,E1 1076.546,E2 1076.546} C_VEL
LIN {X 0,Y 751.76,Z 749.56,A -85,B 0,C 180,E1 1080.003,E2 1080.003} C_VEL
LIN {X 0,Y 751.689,Z 749.56,A -85,B 0,C 180,E1 1084.616,E2 1084.616} C_VEL
LIN {X 0,Y 751.659,Z 749.56,A -85,B 0,C 180,E1 1088.093,E2 1088.093} C_VEL
LIN {X 0,Y 751.587,Z 749.56,A -85,B 0,C 180,E1 1091.602,E2 1091.602} C_VEL
LIN {X 0,Y 751.522,Z 749.56,A -85,B 0,C 180,E1 1095.17,E2 1095.17} C_VEL
LIN {X 0,Y 751.775,Z 749.56,A -85,B 0,C 180,E1 1099.985,E2 1099.985} C_VEL
LIN {X 0,Y 751.703,Z 749.56,A -85,B 0,C 180,E1 1106.252,E2 1106.252} C_VEL
LIN {X 0,Y 751.556,Z 749.56,A -85,B 0,C 180,E1 1111.523,E2 1111.523} C_VEL
LIN {X 0,Y 751.444,Z 749.56,A -85,B 0,C 180,E1 1116.45,E2 1116.45} C_VEL
LIN {X 0,Y 751.701,Z 749.56,A -85,B 0,C 180,E1 1120.191,E2 1120.191} C_VEL
LIN {X 0,Y 751.76,Z 749.56,A -85,B 0,C 180,E1 1125.289,E2 1125.289} C_VEL
LIN {X 0,Y 751.932,Z 750.264,A -85,B 0,C 180,E1 1127.89,E2 1127.89} C_VEL
LIN {X 0,Y 753.651,Z 758.451,A -85,B 0,C 180,E1 1128.066,E2 1128.066} C_VEL
LIN {X 0,Y 753.847,Z 809.251,A -85,B 0,C 180,E1 1128.826,E2 1128.826} C_VEL
LIN {X 0,Y 753.731,Z 857.161,A -85,B 0,C 180,E1 1130.059,E2 1130.059} C_VEL
LIN {X 0,Y 753.322,Z 900.979,A -85,B 0,C 180,E1 1131.676,E2 1131.676} C_VEL
LIN {X 0,Y 753.059,Z 944.543,A -85,B 0,C 180,E1 1133.81,E2 1133.81} C_VEL
LIN {X 0,Y 752.694,Z 986.349,A -85,B 0,C 180,E1 1136.456,E2 1136.456} C_VEL
LIN {X 0,Y 752.373,Z 1022.438,A -85,B 0,C 180,E1 1139.344,E2 1139.344} C_VEL
LIN {X 0,Y 752.146,Z 1052.147,A -85,B 0,C 180,E1 1142.302,E2 1142.302} C_VEL
LIN {X 0,Y 751.972,Z 1077.752,A -85,B 0,C 180,E1 1145.494,E2 1145.494} C_VEL
LIN {X 0,Y 751.988,Z 1098.155,A -85,B 0,C 180,E1 1148.795,E2 1148.795} C_VEL
LIN {X 0,Y 751.844,Z 1113.491,A -85,B 0,C 180,E1 1152.152,E2 1152.152} C_VEL
LIN {X 0,Y 751.912,Z 1123.593,A -85,B 0,C 180,E1 1155.451,E2 1155.451} C_VEL
LIN {X 0,Y 751.887,Z 1128.584,A -85,B 0,C 180,E1 1158.406,E2 1158.406} C_VEL
LIN {X 0,Y 751.987,Z 1129.727,A -85,B 0,C 180,E1 1161.914,E2 1161.914} C_VEL
LIN {X 0,Y 751.817,Z 1125.822,A -85,B 0,C 180,E1 1165.389,E2 1165.389} C_VEL
LIN {X 0,Y 751.772,Z 1116.72,A -85,B 0,C 180,E1 1168.849,E2 1168.849} C_VEL
LIN {X 0,Y 751.828,Z 1103.808,A -85,B 0,C 180,E1 1172.016,E2 1172.016} C_VEL
LIN {X 0,Y 751.893,Z 1086.002,A -85,B 0,C 180,E1 1175.189,E2 1175.189} C_VEL
LIN {X 0,Y 752.034,Z 1061.564,A -85,B 0,C 180,E1 1178.523,E2 1178.523} C_VEL
LIN {X 0,Y 752.22,Z 1034.511,A -85,B 0,C 180,E1 1181.443,E2 1181.443} C_VEL
LIN {X 0,Y 752.571,Z 1000.68,A -85,B 0,C 180,E1 1184.388,E2 1184.388} C_VEL
LIN {X 0,Y 752.919,Z 960.221,A -85,B 0,C 180,E1 1187.183,E2 1187.183} C_VEL
LIN {X 0,Y 753.302,Z 918.113,A -85,B 0,C 180,E1 1189.455,E2 1189.455} C_VEL
LIN {X 0,Y 753.667,Z 876.59,A -85,B 0,C 180,E1 1191.195,E2 1191.195} C_VEL
LIN {X 0,Y 753.955,Z 833.333,A -85,B 0,C 180,E1 1192.521,E2 1192.521} C_VEL
LIN {X 0,Y 754.12,Z 792.512,A -85,B 0,C 180,E1 1193.375,E2 1193.375} C_VEL
LIN {X 0,Y 753.437,Z 754.209,A -85,B 0,C 180,E1 1193.902,E2 1193.902} C_VEL
LIN {X 0,Y 751.834,Z 749.56,A -85,B 0,C 180,E1 1194.079,E2 1194.079} C_VEL
LIN {X 0,Y 751.711,Z 749.56,A -85,B 0,C 180,E1 1198.847,E2 1198.847} C_VEL
LIN {X 0,Y 751.762,Z 749.56,A -85,B 0,C 180,E1 1202.87,E2 1202.87} C_VEL
LIN {X 0,Y 751.796,Z 749.56,A -85,B 0,C 180,E1 1207.086,E2 1207.086} C_VEL
LIN {X 0,Y 751.827,Z 749.56,A -85,B 0,C 180,E1 1213.109,E2 1213.109} C_VEL
LIN {X 0,Y 751.384,Z 749.56,A -85,B 0,C 180,E1 1216.854,E2 1216.854} C_VEL
LIN {X 0,Y 751.629,Z 749.56,A -85,B 0,C 180,E1 1221.441,E2 1221.441} C_VEL
LIN {X 0,Y 751.543,Z 749.56,A -85,B 0,C 180,E1 1225.732,E2 1225.732} C_VEL
LIN {X 0,Y 751.656,Z 749.56,A -85,B 0,C 180,E1 1229.823,E2 1229.823} C_VEL
LIN {X 0,Y 751.463,Z 749.56,A -85,B 0,C 180,E1 1235.016,E2 1235.016} C_VEL
LIN {X 0,Y 751.758,Z 749.56,A -85,B 0,C 180,E1 1240.014,E2 1240.014} C_VEL
LIN {X 0,Y 751.681,Z 749.56,A -85,B 0,C 180,E1 1246.037,E2 1246.037} C_VEL
LIN {X 0,Y 751.703,Z 749.56,A -85,B 0,C 180,E1 1250.742,E2 1250.742} C_VEL
LIN {X 0,Y 751.824,Z 749.56,A -85,B 0,C 180,E1 1254.229,E2 1254.229} C_VEL
LIN {X 0,Y 751.733,Z 749.56,A -85,B 0,C 180,E1 1258.301,E2 1258.301} C_VEL
LIN {X 0,Y 747.743,Z 749.56,A -85,B 0,C 180,E1 1259.607,E2 1259.607} C_VEL
LIN {X 0,Y 744.031,Z 749.56,A -85,B 0,C 180,E1 1260.926,E2 1260.926} C_VEL
LIN {X 0,Y 743.848,Z 749.56,A -85,B 0,C 180,E1 1265.827,E2 1265.827} C_VEL
LIN {X 0,Y 743.733,Z 749.56,A -85,B 0,C 180,E1 1270.534,E2 1270.534} C_VEL
LIN {X 0,Y 743.87,Z 749.56,A -85,B 0,C 180,E1 1275.31,E2 1275.31} C_VEL
LIN {X 0,Y 743.924,Z 749.56,A -85,B 0,C 180,E1 1280.198,E2 1280.198} C_VEL
LIN {X 0,Y 743.747,Z 749.56,A -85,B 0,C 180,E1 1285.254,E2 1285.254} C_VEL
LIN {X 0,Y 743.768,Z 749.56,A -85,B 0,C 180,E1 1289.181,E2 1289.181} C_VEL
LIN {X 0,Y 743.767,Z 749.56,A -85,B 0,C 180,E1 1293.59,E2 1293.59} C_VEL
LIN {X 0,Y 743.762,Z 749.56,A -85,B 0,C 180,E1 1297.591,E2 1297.591} C_VEL
LIN {X 0,Y 743.912,Z 749.56,A -85,B 0,C 180,E1 1303.679,E2 1303.679} C_VEL
LIN {X 0,Y 743.698,Z 749.56,A -85,B 0,C 180,E1 1309.442,E2 1309.442} C_VEL
LIN {X 0,Y 743.938,Z 749.66,A -85,B 0,C 180,E1 1312.414,E2 1312.414} C_VEL
LIN {X 0,Y 747.697,Z 759.942,A -85,B 0,C 180,E1 1312.757,E2 1312.757} C_VEL
LIN {X 0,Y 748.004,Z 847.025,A -85,B 0,C 180,E1 1313.906,E2 1313.906} C_VEL
LIN {X 0,Y 747.428,Z 892.829,A -85,B 0,C 180,E1 1314.955,E2 1314.955} C_VEL
LIN {X 0,Y 746.956,Z 940.165,A -85,B 0,C 180,E1 1316.56,E2 1316.56} C_VEL
LIN {X 0,Y 746.371,Z 986.723,A -85,B 0,C 180,E1 1318.671,E2 1318.671} C_VEL
LIN {X 0,Y 745.786,Z 1028.678,A -85,B 0,C 180,E1 1321.104,E2 1321.104} C_VEL
LIN {X 0,Y 745.189,Z 1069.519,A -85,B 0,C 180,E1 1324.04,E2 1324.04} C_VEL
LIN {X 0,Y 744.684,Z 1106.119,A -85,B 0,C 180,E1 1327.321,E2 1327.321} C_VEL
LIN {X 0,Y 744.358,Z 1135.581,A -85,B 0,C 180,E1 1330.585,E2 1330.585} C_VEL
LIN {X 0,Y 744.102,Z 1160.882,A -85,B 0,C 180,E1 1334.087,E2 1334.087} C_VEL
LIN {X 0,Y 744.02,Z 1179.608,A -85,B 0,C 180,E1 1337.399,E2 1337.399} C_VEL
LIN {X 0,Y 743.99,Z 1194.428,A -85,B 0,C 180,E1 1340.943,E2 1340.943} C_VEL
LIN {X 0,Y 743.965,Z 1204.102,A -85,B 0,C 180,E1 1344.411,E2 1344.411} C_VEL
LIN {X 0,Y 743.985,Z 1208.974,A -85,B 0,C 180,E1 1347.671,E2 1347.671} C_VEL
LIN {X 0,Y 744.125,Z 1209.669,A -85,B 0,C 180,E1 1351.163,E2 1351.163} C_VEL
LIN {X 0,Y 743.867,Z 1205.912,A -85,B 0,C 180,E1 1354.66,E2 1354.66} C_VEL
LIN {X 0,Y 743.848,Z 1197.335,A -85,B 0,C 180,E1 1358.175,E2 1358.175} C_VEL
LIN {X 0,Y 743.928,Z 1185.044,A -85,B 0,C 180,E1 1361.422,E2 1361.422} C_VEL
LIN {X 0,Y 744.076,Z 1166.461,A -85,B 0,C 180,E1 1365.006,E2 1365.006} C_VEL
LIN {X 0,Y 744.249,Z 1144.067,A -85,B 0,C 180,E1 1368.343,E2 1368.343} C_VEL
LIN {X 0,Y 744.582,Z 1115.341,A -85,B 0,C 180,E1 1371.724,E2 1371.724} C_VEL
LIN {X 0,Y 745.038,Z 1082.217,A -85,B 0,C 180,E1 1374.901,E2 1374.901} C_VEL
LIN {X 0,Y 745.61,Z 1041.443,A -85,B 0,C 180,E1 1378.048,E2 1378.048} C_VEL
LIN {X 0,Y 746.189,Z 999.737,A -85,B 0,C 180,E1 1380.628,E2 1380.628} C_VEL
LIN {X 0,Y 746.868,Z 956.091,A -85,B 0,C 180,E1 1382.779,E2 1382.779} C_VEL
LIN {X 0,Y 747.407,Z 912.528,A -85,B 0,C 180,E1 1384.432,E2 1384.432} C_VEL
LIN {X 0,Y 747.81,Z 867.424,A -85,B 0,C 180,E1 1385.682,E2 1385.682} C_VEL
LIN {X 0,Y 748.073,Z 823.017,A -85,B 0,C 180,E1 1386.472,E2 1386.472} C_VEL
LIN {X 0,Y 747.125,Z 757.103,A -85,B 0,C 180,E1 1387.31,E2 1387.31} C_VEL
LIN {X 0,Y 743.932,Z 749.56,A -85,B 0,C 180,E1 1387.612,E2 1387.612} C_VEL
LIN {X 0,Y 743.918,Z 749.56,A -85,B 0,C 180,E1 1393.68,E2 1393.68} C_VEL
LIN {X 0,Y 743.523,Z 749.56,A -85,B 0,C 180,E1 1398.762,E2 1398.762} C_VEL
LIN {X 0,Y 743.555,Z 749.56,A -85,B 0,C 180,E1 1402.436,E2 1402.436} C_VEL
LIN {X 0,Y 743.534,Z 749.56,A -85,B 0,C 180,E1 1406.723,E2 1406.723} C_VEL
LIN {X 0,Y 743.575,Z 749.56,A -85,B 0,C 180,E1 1410.91,E2 1410.91} C_VEL
LIN {X 0,Y 743.675,Z 749.56,A -85,B 0,C 180,E1 1414.744,E2 1414.744} C_VEL
LIN {X 0,Y 743.67,Z 749.56,A -85,B 0,C 180,E1 1419.794,E2 1419.794} C_VEL
LIN {X 0,Y 743.856,Z 749.56,A -85,B 0,C 180,E1 1424.69,E2 1424.69} C_VEL
LIN {X 0,Y 743.741,Z 749.56,A -85,B 0,C 180,E1 1429.467,E2 1429.467} C_VEL
LIN {X 0,Y 743.839,Z 749.56,A -85,B 0,C 180,E1 1434.173,E2 1434.173} C_VEL
LIN {X 0,Y 744.064,Z 749.56,A -85,B 0,C 180,E1 1438.839,E2 1438.839} C_VEL
LIN {X 0,Y 743.953,Z 749.56,A -85,B 0,C 180,E1 1443.497,E2 1443.497} C_VEL
LIN {X 0,Y 743.753,Z 749.56,A -85,B 0,C 180,E1 1448.18,E2 1448.18} C_VEL
LIN {X 0,Y 743.668,Z 749.56,A -85,B 0,C 180,E1 1451.728,E2 1451.728} C_VEL
LIN {X 0,Y 743.605,Z 749.56,A -85,B 0,C 180,E1 1455.322,E2 1455.322} C_VEL
LIN {X 0,Y 743.646,Z 749.56,A -85,B 0,C 180,E1 1460.815,E2 1460.815} C_VEL
LIN {X 0,Y 743.684,Z 749.56,A -85,B 0,C 180,E1 1466.614,E2 1466.614} C_VEL
LIN {X 0,Y 743.581,Z 749.56,A -85,B 0,C 180,E1 1471.901,E2 1471.901} C_VEL
LIN {X 0,Y 743.598,Z 749.56,A -85,B 0,C 180,E1 1476.115,E2 1476.115} C_VEL
LIN {X 0,Y 743.69,Z 749.56,A -85,B 0,C 180,E1 1480.563,E2 1480.563} C_VEL
LIN {X 0,Y 743.856,Z 749.56,A -85,B 0,C 180,E1 1485.324,E2 1485.324} C_VEL
LIN {X 0,Y 743.972,Z 749.56,A -85,B 0,C 180,E1 1487.463,E2 1487.463} C_VEL
LIN {X 0,Y 746.981,Z 758.521,A -85,B 0,C 180,E1 1487.735,E2 1487.735} C_VEL
LIN {X 0,Y 747.114,Z 809.918,A -85,B 0,C 180,E1 1488.516,E2 1488.516} C_VEL
LIN {X 0,Y 746.862,Z 857.813,A -85,B 0,C 180,E1 1489.763,E2 1489.763} C_VEL
LIN {X 0,Y 746.273,Z 901.617,A -85,B 0,C 180,E1 1491.4,E2 1491.4} C_VEL
LIN {X 0,Y 745.775,Z 945.25,A -85,B 0,C 180,E1 1493.565,E2 1493.565} C_VEL
LIN {X 0,Y 745.222,Z 987.128,A -85,B 0,C 180,E1 1496.249,E2 1496.249} C_VEL
LIN {X 0,Y 744.732,Z 1023.989,A -85,B 0,C 180,E1 1499.249,E2 1499.249} C_VEL
LIN {X 0,Y 744.377,Z 1054.059,A -85,B 0,C 180,E1 1502.319,E2 1502.319} C_VEL
LIN {X 0,Y 744.147,Z 1079.402,A -85,B 0,C 180,E1 1505.56,E2 1505.56} C_VEL
LIN {X 0,Y 744.064,Z 1100.5,A -85,B 0,C 180,E1 1509.115,E2 1509.115} C_VEL
LIN {X 0,Y 743.938,Z 1114.289,A -85,B 0,C 180,E1 1512.261,E2 1512.261} C_VEL
LIN {X 0,Y 743.936,Z 1124.624,A -85,B 0,C 180,E1 1515.893,E2 1515.893} C_VEL
LIN {X 0,Y 743.875,Z 1129.531,A -85,B 0,C 180,E1 1519.466,E2 1519.466} C_VEL
LIN {X 0,Y 744.111,Z 1129.044,A -85,B 0,C 180,E1 1523.002,E2 1523.002} C_VEL
LIN {X 0,Y 744.084,Z 1123.613,A -85,B 0,C 180,E1 1526.508,E2 1526.508} C_VEL
LIN {X 0,Y 744.19,Z 1111.764,A -85,B 0,C 180,E1 1530.291,E2 1530.291} C_VEL
LIN {X 0,Y 744.135,Z 1095.304,A -85,B 0,C 180,E1 1533.785,E2 1533.785} C_VEL
LIN {X 0,Y 744.31,Z 1071.534,A -85,B 0,C 180,E1 1537.437,E2 1537.437} C_VEL
LIN {X 0,Y 744.503,Z 1044.187,A -85,B 0,C 180,E1 1540.674,E2 1540.674} C_VEL
LIN {X 0,Y 744.925,Z 1012.773,A -85,B 0,C 180,E1 1543.649,E2 1543.649} C_VEL
LIN {X 0,Y 745.446,Z 974.161,A -85,B 0,C 180,E1 1546.563,E2 1546.563} C_VEL
LIN {X 0,Y 745.956,Z 932.439,A -85,B 0,C 180,E1 1549.038,E2 1549.038} C_VEL
LIN {X 0,Y 746.503,Z 891.126,A -85,B 0,C 180,E1 1550.946,E2 1550.946} C_VEL
LIN {X 0,Y 746.977,Z 846.514,A -85,B 0,C 180,E1 1552.487,E2 1552.487} C_VEL
LIN {X 0,Y 747.276,Z 800.953,A -85,B 0,C 180,E1 1553.56,E2 1553.56} C_VEL
LIN {X 0,Y 746.652,Z 756.807,A -85,B 0,C 180,E1 1554.211,E2 1554.211} C_VEL
LIN {X 0,Y 743.799,Z 749.56,A -85,B 0,C 180,E1 1554.506,E2 1554.506} C_VEL
LIN {X 0,Y 743.74,Z 749.56,A -85,B 0,C 180,E1 1559.186,E2 1559.186} C_VEL
LIN {X 0,Y 743.681,Z 749.56,A -85,B 0,C 180,E1 1563.573,E2 1563.573} C_VEL
LIN {X 0,Y 743.749,Z 749.56,A -85,B 0,C 180,E1 1567.583,E2 1567.583} C_VEL
LIN {X 0,Y 743.908,Z 749.56,A -85,B 0,C 180,E1 1573,E2 1573} C_VEL
LIN {X 0,Y 743.458,Z 749.56,A -85,B 0,C 180,E1 1577.032,E2 1577.032} C_VEL
LIN {X 0,Y 743.714,Z 749.56,A -85,B 0,C 180,E1 1580.954,E2 1580.954} C_VEL
LIN {X 0,Y 743.667,Z 749.56,A -85,B 0,C 180,E1 1585.317,E2 1585.317} C_VEL
LIN {X 0,Y 743.682,Z 749.56,A -85,B 0,C 180,E1 1589.465,E2 1589.465} C_VEL
LIN {X 0,Y 743.649,Z 749.56,A -85,B 0,C 180,E1 1594.736,E2 1594.736} C_VEL
LIN {X 0,Y 743.774,Z 749.56,A -85,B 0,C 180,E1 1599.791,E2 1599.791} C_VEL
LIN {X 0,Y 743.745,Z 749.56,A -85,B 0,C 180,E1 1605.885,E2 1605.885} C_VEL
LIN {X 0,Y 743.846,Z 749.56,A -85,B 0,C 180,E1 1610.643,E2 1610.643} C_VEL
LIN {X 0,Y 743.882,Z 749.56,A -85,B 0,C 180,E1 1614.502,E2 1614.502} C_VEL
LIN {X 0,Y 743.774,Z 749.56,A -85,B 0,C 180,E1 1618.833,E2 1618.833} C_VEL
LIN {X 0,Y 744.031,Z 749.56,A -85,B 0,C 180,E1 1620.926,E2 1620.926} C_VEL
LIN {X 0,Y 741.55,Z 749.56,A -85,B 0,C 180,E1 1621.917,E2 1621.917} C_VEL
LIN {X 0,Y 736.045,Z 749.56,A -85,B 0,C 180,E1 1623.396,E2 1623.396} C_VEL
LIN {X 0,Y 735.957,Z 749.56,A -85,B 0,C 180,E1 1623.567,E2 1623.567} C_VEL
LIN {X 0,Y 736.041,Z 749.56,A -85,B 0,C 180,E1 1628.26,E2 1628.26} C_VEL
LIN {X 0,Y 735.936,Z 749.56,A -85,B 0,C 180,E1 1633.051,E2 1633.051} C_VEL
LIN {X 0,Y 735.847,Z 749.56,A -85,B 0,C 180,E1 1637.938,E2 1637.938} C_VEL
LIN {X 0,Y 735.824,Z 749.56,A -85,B 0,C 180,E1 1642.459,E2 1642.459} C_VEL
LIN {X 0,Y 735.78,Z 749.56,A -85,B 0,C 180,E1 1646.858,E2 1646.858} C_VEL
LIN {X 0,Y 735.912,Z 749.56,A -85,B 0,C 180,E1 1652.265,E2 1652.265} C_VEL
LIN {X 0,Y 735.801,Z 749.56,A -85,B 0,C 180,E1 1656.778,E2 1656.778} C_VEL
LIN {X 0,Y 735.946,Z 749.56,A -85,B 0,C 180,E1 1662.653,E2 1662.653} C_VEL
LIN {X 0,Y 735.57,Z 749.56,A -85,B 0,C 180,E1 1667.316,E2 1667.316} C_VEL
LIN {X 0,Y 735.977,Z 749.729,A -85,B 0,C 180,E1 1671.936,E2 1671.936} C_VEL
LIN {X 0,Y 741.41,Z 761.57,A -85,B 0,C 180,E1 1672.406,E2 1672.406} C_VEL
LIN {X 0,Y 741.618,Z 847.001,A -85,B 0,C 180,E1 1673.545,E2 1673.545} C_VEL
LIN {X 0,Y 740.88,Z 892.604,A -85,B 0,C 180,E1 1674.593,E2 1674.593} C_VEL
LIN {X 0,Y 740.191,Z 940.169,A -85,B 0,C 180,E1 1676.214,E2 1676.214} C_VEL
LIN {X 0,Y 739.321,Z 987.951,A -85,B 0,C 180,E1 1678.4,E2 1678.4} C_VEL
LIN {X 0,Y 738.505,Z 1031.324,A -85,B 0,C 180,E1 1680.969,E2 1680.969} C_VEL
LIN {X 0,Y 737.72,Z 1070.617,A -85,B 0,C 180,E1 1683.85,E2 1683.85} C_VEL
LIN {X 0,Y 737.056,Z 1108.441,A -85,B 0,C 180,E1 1687.304,E2 1687.304} C_VEL
LIN {X 0,Y 736.559,Z 1138.024,A -85,B 0,C 180,E1 1690.683,E2 1690.683} C_VEL
LIN {X 0,Y 736.283,Z 1162.852,A -85,B 0,C 180,E1 1694.22,E2 1694.22} C_VEL
LIN {X 0,Y 736.086,Z 1181.274,A -85,B 0,C 180,E1 1697.615,E2 1697.615} C_VEL
LIN {X 0,Y 736.052,Z 1195.442,A -85,B 0,C 180,E1 1701.142,E2 1701.142} C_VEL
LIN {X 0,Y 736.032,Z 1204.59,A -85,B 0,C 180,E1 1704.59,E2 1704.59} C_VEL
LIN {X 0,Y 736.091,Z 1208.971,A -85,B 0,C 180,E1 1707.646,E2 1707.646} C_VEL
LIN {X 0,Y 736.23,Z 1209.669,A -85,B 0,C 180,E1 1711.176,E2 1711.176} C_VEL
LIN {X 0,Y 735.982,Z 1205.912,A -85,B 0,C 180,E1 1714.71,E2 1714.71} C_VEL
LIN {X 0,Y 735.952,Z 1197.334,A -85,B 0,C 180,E1 1718.263,E2 1718.263} C_VEL
LIN {X 0,Y 736.029,Z 1185.045,A -85,B 0,C 180,E1 1721.547,E2 1721.547} C_VEL
LIN {X 0,Y 736.225,Z 1167.317,A -85,B 0,C 180,E1 1725.022,E2 1725.022} C_VEL
LIN {X 0,Y 736.45,Z 1145.171,A -85,B 0,C 180,E1 1728.389,E2 1728.389} C_VEL
LIN {X 0,Y 736.904,Z 1116.954,A -85,B 0,C 180,E1 1731.789,E2 1731.789} C_VEL
LIN {X 0,Y 737.515,Z 1082.37,A -85,B 0,C 180,E1 1735.16,E2 1735.16} C_VEL
LIN {X 0,Y 738.292,Z 1041.488,A -85,B 0,C 180,E1 1738.348,E2 1738.348} C_VEL
LIN {X 0,Y 739.097,Z 1000.539,A -85,B 0,C 180,E1 1740.909,E2 1740.909} C_VEL
LIN {X 0,Y 740.013,Z 957.097,A -85,B 0,C 180,E1 1743.075,E2 1743.075} C_VEL
LIN {X 0,Y 740.763,Z 913.103,A -85,B 0,C 180,E1 1744.767,E2 1744.767} C_VEL
LIN {X 0,Y 741.318,Z 868.916,A -85,B 0,C 180,E1 1746.008,E2 1746.008} C_VEL
LIN {X 0,Y 741.727,Z 822.462,A -85,B 0,C 180,E1 1746.842,E2 1746.842} C_VEL
LIN {X 0,Y 740.995,Z 760.164,A -85,B 0,C 180,E1 1747.635,E2 1747.635} C_VEL
LIN {X 0,Y 736.036,Z 751.18,A -85,B 0,C 180,E1 1748.042,E2 1748.042} C_VEL
LIN {X 0,Y 735.822,Z 749.56,A -85,B 0,C 180,E1 1748.124,E2 1748.124} C_VEL
LIN {X 0,Y 736.005,Z 749.56,A -85,B 0,C 180,E1 1754.064,E2 1754.064} C_VEL
LIN {X 0,Y 735.797,Z 749.56,A -85,B 0,C 180,E1 1759.453,E2 1759.453} C_VEL
LIN {X 0,Y 735.76,Z 749.56,A -85,B 0,C 180,E1 1764.898,E2 1764.898} C_VEL
LIN {X 0,Y 735.679,Z 749.56,A -85,B 0,C 180,E1 1770.467,E2 1770.467} C_VEL
LIN {X 0,Y 735.78,Z 749.56,A -85,B 0,C 180,E1 1774.642,E2 1774.642} C_VEL
LIN {X 0,Y 735.768,Z 749.56,A -85,B 0,C 180,E1 1779.568,E2 1779.568} C_VEL
LIN {X 0,Y 735.924,Z 749.56,A -85,B 0,C 180,E1 1784.813,E2 1784.813} C_VEL
LIN {X 0,Y 735.847,Z 749.56,A -85,B 0,C 180,E1 1789.352,E2 1789.352} C_VEL
LIN {X 0,Y 735.929,Z 749.56,A -85,B 0,C 180,E1 1794.11,E2 1794.11} C_VEL
LIN {X 0,Y 736.17,Z 749.56,A -85,B 0,C 180,E1 1798.827,E2 1798.827} C_VEL
LIN {X 0,Y 736.042,Z 749.56,A -85,B 0,C 180,E1 1803.535,E2 1803.535} C_VEL
LIN {X 0,Y 735.85,Z 749.56,A -85,B 0,C 180,E1 1808.268,E2 1808.268} C_VEL
LIN {X 0,Y 735.77,Z 749.56,A -85,B 0,C 180,E1 1811.855,E2 1811.855} C_VEL
LIN {X 0,Y 735.672,Z 749.56,A -85,B 0,C 180,E1 1815.491,E2 1815.491} C_VEL
LIN {X 0,Y 735.847,Z 749.56,A -85,B 0,C 180,E1 1820.437,E2 1820.437} C_VEL
LIN {X 0,Y 735.712,Z 749.56,A -85,B 0,C 180,E1 1825.556,E2 1825.556} C_VEL
LIN {X 0,Y 735.783,Z 749.56,A -85,B 0,C 180,E1 1830.898,E2 1830.898} C_VEL
LIN {X 0,Y 735.761,Z 749.56,A -85,B 0,C 180,E1 1835.11,E2 1835.11} C_VEL
LIN {X 0,Y 735.79,Z 749.56,A -85,B 0,C 180,E1 1840.547,E2 1840.547} C_VEL
LIN {X 0,Y 735.939,Z 749.56,A -85,B 0,C 180,E1 1845.951,E2 1845.951} C_VEL
LIN {X 0,Y 736.002,Z 749.56,A -85,B 0,C 180,E1 1847.047,E2 1847.047} C_VEL
LIN {X 0,Y 740.45,Z 762.106,A -85,B 0,C 180,E1 1847.445,E2 1847.445} C_VEL
LIN {X 0,Y 740.332,Z 812.245,A -85,B 0,C 180,E1 1848.233,E2 1848.233} C_VEL
LIN {X 0,Y 740.006,Z 860.004,A -85,B 0,C 180,E1 1849.509,E2 1849.509} C_VEL
LIN {X 0,Y 739.163,Z 906.392,A -85,B 0,C 180,E1 1851.301,E2 1851.301} C_VEL
LIN {X 0,Y 738.454,Z 947.971,A -85,B 0,C 180,E1 1853.432,E2 1853.432} C_VEL
LIN {X 0,Y 737.733,Z 988.542,A -85,B 0,C 180,E1 1856.086,E2 1856.086} C_VEL
LIN {X 0,Y 737.116,Z 1025.72,A -85,B 0,C 180,E1 1859.169,E2 1859.169} C_VEL
LIN {X 0,Y 736.557,Z 1057.643,A -85,B 0,C 180,E1 1862.529,E2 1862.529} C_VEL
LIN {X 0,Y 736.272,Z 1081.822,A -85,B 0,C 180,E1 1865.766,E2 1865.766} C_VEL
LIN {X 0,Y 736.164,Z 1101.75,A -85,B 0,C 180,E1 1869.229,E2 1869.229} C_VEL
LIN {X 0,Y 736.004,Z 1115.536,A -85,B 0,C 180,E1 1872.526,E2 1872.526} C_VEL
LIN {X 0,Y 736.057,Z 1124.421,A -85,B 0,C 180,E1 1875.738,E2 1875.738} C_VEL
LIN {X 0,Y 735.974,Z 1129.447,A -85,B 0,C 180,E1 1879.352,E2 1879.352} C_VEL
LIN {X 0,Y 736.199,Z 1129.129,A -85,B 0,C 180,E1 1882.926,E2 1882.926} C_VEL
LIN {X 0,Y 736.18,Z 1123.811,A -85,B 0,C 180,E1 1886.47,E2 1886.47} C_VEL
LIN {X 0,Y 736.209,Z 1113.284,A -85,B 0,C 180,E1 1890.001,E2 1890.001} C_VEL
LIN {X 0,Y 736.276,Z 1095.861,A -85,B 0,C 180,E1 1893.825,E2 1893.825} C_VEL
LIN {X 0,Y 736.486,Z 1072.256,A -85,B 0,C 180,E1 1897.517,E2 1897.517} C_VEL
LIN {X 0,Y 736.786,Z 1045.15,A -85,B 0,C 180,E1 1900.787,E2 1900.787} C_VEL
LIN {X 0,Y 737.349,Z 1012.303,A -85,B 0,C 180,E1 1903.935,E2 1903.935} C_VEL
LIN {X 0,Y 738.035,Z 974.921,A -85,B 0,C 180,E1 1906.786,E2 1906.786} C_VEL
LIN {X 0,Y 738.735,Z 933.419,A -85,B 0,C 180,E1 1909.283,E2 1909.283} C_VEL
LIN {X 0,Y 739.51,Z 891.976,A -85,B 0,C 180,E1 1911.225,E2 1911.225} C_VEL
LIN {X 0,Y 740.137,Z 847.378,A -85,B 0,C 180,E1 1912.786,E2 1912.786} C_VEL
LIN {X 0,Y 740.587,Z 802.263,A -85,B 0,C 180,E1 1913.869,E2 1913.869} C_VEL
LIN {X 0,Y 740.156,Z 759.523,A -85,B 0,C 180,E1 1914.51,E2 1914.51} C_VEL
LIN {X 0,Y 735.8,Z 749.56,A -85,B 0,C 180,E1 1914.854,E2 1914.854} C_VEL
LIN {X 0,Y 735.757,Z 749.56,A -85,B 0,C 180,E1 1919.533,E2 1919.533} C_VEL
LIN {X 0,Y 735.764,Z 749.56,A -85,B 0,C 180,E1 1923.679,E2 1923.679} C_VEL
LIN {X 0,Y 735.581,Z 749.56,A -85,B 0,C 180,E1 1928.673,E2 1928.673} C_VEL
LIN {X 0,Y 735.979,Z 749.56,A -85,B 0,C 180,E1 1934.053,E2 1934.053} C_VEL
LIN {X 0,Y 735.793,Z 749.56,A -85,B 0,C 180,E1 1939.455,E2 1939.455} C_VEL
LIN {X 0,Y 735.768,Z 749.56,A -85,B 0,C 180,E1 1945.239,E2 1945.239} C_VEL
LIN {X 0,Y 735.662,Z 749.56,A -85,B 0,C 180,E1 1950.459,E2 1950.459} C_VEL
LIN {X 0,Y 735.748,Z 749.56,A -85,B 0,C 180,E1 1954.65,E2 1954.65} C_VEL
LIN {X 0,Y 735.835,Z 749.56,A -85,B 0,C 180,E1 1959.563,E2 1959.563} C_VEL
LIN {X 0,Y 735.81,Z 749.56,A -85,B 0,C 180,E1 1965.729,E2 1965.729} C_VEL
LIN {X 0,Y 735.952,Z 749.56,A -85,B 0,C 180,E1 1970.542,E2 1970.542} C_VEL
LIN {X 0,Y 736.044,Z 749.56,A -85,B 0,C 180,E1 1974.105,E2 1974.105} C_VEL
LIN {X 0,Y 735.905,Z 749.56,A -85,B 0,C 180,E1 1978.82,E2 1978.82} C_VEL
LIN {X 0,Y 735.928,Z 749.56,A -85,B 0,C 180,E1 1982.35,E2 1982.35} C_VEL
LIN {X 0,Y 735.957,Z 749.56,A -85,B 0,C 180,E1 1983.567,E2 1983.567} C_VEL
LIN {X 0,Y 734.735,Z 749.56,A -85,B 0,C 180,E1 1984.241,E2 1984.241} C_VEL
LIN {X 0,Y 728.114,Z 749.56,A -85,B 0,C 180,E1 1986.073,E2 1986.073} C_VEL
LIN {X 0,Y 728.006,Z 749.56,A -85,B 0,C 180,E1 1986.246,E2 1986.246} C_VEL
LIN {X 0,Y 727.942,Z 749.56,A -85,B 0,C 180,E1 1990.765,E2 1990.765} C_VEL
LIN {X 0,Y 728.07,Z 749.56,A -85,B 0,C 180,E1 1995.65,E2 1995.65} C_VEL
LIN {X 0,Y 727.975,Z 749.56,A -85,B 0,C 180,E1 2000.914,E2 2000.914} C_VEL
LIN {X 0,Y 727.863,Z 749.56,A -85,B 0,C 180,E1 2005.845,E2 2005.845} C_VEL
LIN {X 0,Y 727.865,Z 749.56,A -85,B 0,C 180,E1 2009.882,E2 2009.882} C_VEL
LIN {X 0,Y 727.891,Z 749.56,A -85,B 0,C 180,E1 2014.089,E2 2014.089} C_VEL
LIN {X 0,Y 727.735,Z 749.56,A -85,B 0,C 180,E1 2018.528,E2 2018.528} C_VEL
LIN {X 0,Y 728.022,Z 749.56,A -85,B 0,C 180,E1 2023.407,E2 2023.407} C_VEL
LIN {X 0,Y 727.682,Z 749.56,A -85,B 0,C 180,E1 2028.378,E2 2028.378} C_VEL
LIN {X 0,Y 728.067,Z 749.722,A -85,B 0,C 180,E1 2031.447,E2 2031.447} C_VEL
LIN {X 0,Y 734.906,Z 763.888,A -85,B 0,C 180,E1 2032.043,E2 2032.043} C_VEL
LIN {X 0,Y 735.224,Z 848.213,A -85,B 0,C 180,E1 2033.199,E2 2033.199} C_VEL
LIN {X 0,Y 734.323,Z 894.299,A -85,B 0,C 180,E1 2034.277,E2 2034.277} C_VEL
LIN {X 0,Y 733.397,Z 942.093,A -85,B 0,C 180,E1 2035.939,E2 2035.939} C_VEL
LIN {X 0,Y 732.335,Z 987.747,A -85,B 0,C 180,E1 2038.053,E2 2038.053} C_VEL
LIN {X 0,Y 731.334,Z 1030.637,A -85,B 0,C 180,E1 2040.61,E2 2040.61} C_VEL
LIN {X 0,Y 730.347,Z 1068.911,A -85,B 0,C 180,E1 2043.42,E2 2043.42} C_VEL
LIN {X 0,Y 729.513,Z 1106.122,A -85,B 0,C 180,E1 2046.823,E2 2046.823} C_VEL
LIN {X 0,Y 728.887,Z 1135.57,A -85,B 0,C 180,E1 2050.154,E2 2050.154} C_VEL
LIN {X 0,Y 728.498,Z 1160.885,A -85,B 0,C 180,E1 2053.737,E2 2053.737} C_VEL
LIN {X 0,Y 728.326,Z 1179.955,A -85,B 0,C 180,E1 2057.192,E2 2057.192} C_VEL
LIN {X 0,Y 728.18,Z 1195.443,A -85,B 0,C 180,E1 2061.045,E2 2061.045} C_VEL
LIN {X 0,Y 728.257,Z 1203.568,A -85,B 0,C 180,E1 2064.044,E2 2064.044} C_VEL
LIN {X 0,Y 728.188,Z 1208.969,A -85,B 0,C 180,E1 2067.621,E2 2067.621} C_VEL
LIN {X 0,Y 728.328,Z 1209.669,A -85,B 0,C 180,E1 2071.188,E2 2071.188} C_VEL
LIN {X 0,Y 728.084,Z 1205.478,A -85,B 0,C 180,E1 2074.997,E2 2074.997} C_VEL
LIN {X 0,Y 728.063,Z 1197.334,A -85,B 0,C 180,E1 2078.353,E2 2078.353} C_VEL
LIN {X 0,Y 728.156,Z 1185.046,A -85,B 0,C 180,E1 2081.673,E2 2081.673} C_VEL
LIN {X 0,Y 728.392,Z 1167.73,A -85,B 0,C 180,E1 2085.116,E2 2085.116} C_VEL
LIN {X 0,Y 728.665,Z 1145.172,A -85,B 0,C 180,E1 2088.593,E2 2088.593} C_VEL
LIN {X 0,Y 729.228,Z 1117.087,A -85,B 0,C 180,E1 2092.016,E2 2092.016} C_VEL
LIN {X 0,Y 730.038,Z 1082.369,A -85,B 0,C 180,E1 2095.436,E2 2095.436} C_VEL
LIN {X 0,Y 731.011,Z 1041.486,A -85,B 0,C 180,E1 2098.656,E2 2098.656} C_VEL
LIN {X 0,Y 732.076,Z 1000.192,A -85,B 0,C 180,E1 2101.259,E2 2101.259} C_VEL
LIN {X 0,Y 733.209,Z 956.371,A -85,B 0,C 180,E1 2103.455,E2 2103.455} C_VEL
LIN {X 0,Y 734.168,Z 913.03,A -85,B 0,C 180,E1 2105.127,E2 2105.127} C_VEL
LIN {X 0,Y 734.857,Z 869.375,A -85,B 0,C 180,E1 2106.364,E2 2106.364} C_VEL
LIN {X 0,Y 735.377,Z 824.012,A -85,B 0,C 180,E1 2107.192,E2 2107.192} C_VEL
LIN {X 0,Y 734.571,Z 763.338,A -85,B 0,C 180,E1 2107.984,E2 2107.984} C_VEL
LIN {X 0,Y 727.97,Z 751.211,A -85,B 0,C 180,E1 2108.54,E2 2108.54} C_VEL
LIN {X 0,Y 727.782,Z 749.56,A -85,B 0,C 180,E1 2108.605,E2 2108.605} C_VEL
LIN {X 0,Y 728.025,Z 749.56,A -85,B 0,C 180,E1 2113.411,E2 2113.411} C_VEL
LIN {X 0,Y 727.674,Z 749.56,A -85,B 0,C 180,E1 2118.382,E2 2118.382} C_VEL
LIN {X 0,Y 727.754,Z 749.56,A -85,B 0,C 180,E1 2122.978,E2 2122.978} C_VEL
LIN {X 0,Y 727.715,Z 749.56,A -85,B 0,C 180,E1 2127.326,E2 2127.326} C_VEL
LIN {X 0,Y 727.688,Z 749.56,A -85,B 0,C 180,E1 2131.473,E2 2131.473} C_VEL
LIN {X 0,Y 727.737,Z 749.56,A -85,B 0,C 180,E1 2136.013,E2 2136.013} C_VEL
LIN {X 0,Y 727.813,Z 749.56,A -85,B 0,C 180,E1 2140.601,E2 2140.601} C_VEL
LIN {X 0,Y 728.05,Z 749.56,A -85,B 0,C 180,E1 2144.349,E2 2144.349} C_VEL
LIN {X 0,Y 727.944,Z 749.56,A -85,B 0,C 180,E1 2149.235,E2 2149.235} C_VEL
LIN {X 0,Y 728.037,Z 749.56,A -85,B 0,C 180,E1 2154.046,E2 2154.046} C_VEL
LIN {X 0,Y 728.263,Z 749.56,A -85,B 0,C 180,E1 2158.814,E2 2158.814} C_VEL
LIN {X 0,Y 728.131,Z 749.56,A -85,B 0,C 180,E1 2163.573,E2 2163.573} C_VEL
LIN {X 0,Y 727.962,Z 749.56,A -85,B 0,C 180,E1 2168.359,E2 2168.359} C_VEL
LIN {X 0,Y 727.845,Z 749.56,A -85,B 0,C 180,E1 2172.634,E2 2172.634} C_VEL
LIN {X 0,Y 727.551,Z 749.56,A -85,B 0,C 180,E1 2177.174,E2 2177.174} C_VEL
LIN {X 0,Y 727.826,Z 749.56,A -85,B 0,C 180,E1 2180.887,E2 2180.887} C_VEL
LIN {X 0,Y 727.823,Z 749.56,A -85,B 0,C 180,E1 2186.777,E2 2186.777} C_VEL
LIN {X 0,Y 727.745,Z 749.56,A -85,B 0,C 180,E1 2191.643,E2 2191.643} C_VEL
LIN {X 0,Y 727.74,Z 749.56,A -85,B 0,C 180,E1 2195.923,E2 2195.923} C_VEL
LIN {X 0,Y 727.919,Z 749.56,A -85,B 0,C 180,E1 2200.062,E2 2200.062} C_VEL
LIN {X 0,Y 727.952,Z 749.56,A -85,B 0,C 180,E1 2205.107,E2 2205.107} C_VEL
LIN {X 0,Y 728.096,Z 750.19,A -85,B 0,C 180,E1 2206.659,E2 2206.659} C_VEL
LIN {X 0,Y 733.914,Z 764.369,A -85,B 0,C 180,E1 2207.132,E2 2207.132} C_VEL
LIN {X 0,Y 733.654,Z 814.24,A -85,B 0,C 180,E1 2207.942,E2 2207.942} C_VEL
LIN {X 0,Y 733.123,Z 860.621,A -85,B 0,C 180,E1 2209.201,E2 2209.201} C_VEL
LIN {X 0,Y 732.09,Z 907.003,A -85,B 0,C 180,E1 2211.013,E2 2211.013} C_VEL
LIN {X 0,Y 731.19,Z 948.682,A -85,B 0,C 180,E1 2213.179,E2 2213.179} C_VEL
LIN {X 0,Y 730.339,Z 988.004,A -85,B 0,C 180,E1 2215.775,E2 2215.775} C_VEL
LIN {X 0,Y 729.519,Z 1025.476,A -85,B 0,C 180,E1 2218.908,E2 2218.908} C_VEL
LIN {X 0,Y 728.856,Z 1056.992,A -85,B 0,C 180,E1 2222.251,E2 2222.251} C_VEL
LIN {X 0,Y 728.468,Z 1081.122,A -85,B 0,C 180,E1 2225.489,E2 2225.489} C_VEL
LIN {X 0,Y 728.315,Z 1101.378,A -85,B 0,C 180,E1 2229.027,E2 2229.027} C_VEL
LIN {X 0,Y 728.148,Z 1115.319,A -85,B 0,C 180,E1 2232.366,E2 2232.366} C_VEL
LIN {X 0,Y 728.191,Z 1124.218,A -85,B 0,C 180,E1 2235.581,E2 2235.581} C_VEL
LIN {X 0,Y 728.068,Z 1129.362,A -85,B 0,C 180,E1 2239.235,E2 2239.235} C_VEL
LIN {X 0,Y 728.287,Z 1129.213,A -85,B 0,C 180,E1 2242.849,E2 2242.849} C_VEL
LIN {X 0,Y 728.276,Z 1124.01,A -85,B 0,C 180,E1 2246.432,E2 2246.432} C_VEL
LIN {X 0,Y 728.315,Z 1113.663,A -85,B 0,C 180,E1 2250.001,E2 2250.001} C_VEL
LIN {X 0,Y 728.406,Z 1096.374,A -85,B 0,C 180,E1 2253.867,E2 2253.867} C_VEL
LIN {X 0,Y 728.697,Z 1074.036,A -85,B 0,C 180,E1 2257.448,E2 2257.448} C_VEL
LIN {X 0,Y 729.083,Z 1047.511,A -85,B 0,C 180,E1 2260.751,E2 2260.751} C_VEL
LIN {X 0,Y 729.793,Z 1013.546,A -85,B 0,C 180,E1 2264.082,E2 2264.082} C_VEL
LIN {X 0,Y 730.647,Z 974.125,A -85,B 0,C 180,E1 2267.123,E2 2267.123} C_VEL
LIN {X 0,Y 731.649,Z 932.066,A -85,B 0,C 180,E1 2269.658,E2 2269.658} C_VEL
LIN {X 0,Y 732.536,Z 891.007,A -85,B 0,C 180,E1 2271.584,E2 2271.584} C_VEL
LIN {X 0,Y 733.402,Z 846.466,A -85,B 0,C 180,E1 2273.142,E2 2273.142} C_VEL
LIN {X 0,Y 733.956,Z 801.849,A -85,B 0,C 180,E1 2274.212,E2 2274.212} C_VEL
LIN {X 0,Y 733.694,Z 762.799,A -85,B 0,C 180,E1 2274.807,E2 2274.807} C_VEL
LIN {X 0,Y 727.843,Z 749.56,A -85,B 0,C 180,E1 2275.302,E2 2275.302} C_VEL
LIN {X 0,Y 727.837,Z 749.56,A -85,B 0,C 180,E1 2279.887,E2 2279.887} C_VEL
LIN {X 0,Y 727.821,Z 749.56,A -85,B 0,C 180,E1 2284.097,E2 2284.097} C_VEL
LIN {X 0,Y 727.705,Z 749.56,A -85,B 0,C 180,E1 2288.534,E2 2288.534} C_VEL
LIN {X 0,Y 728.014,Z 749.56,A -85,B 0,C 180,E1 2293.401,E2 2293.401} C_VEL
LIN {X 0,Y 727.681,Z 749.56,A -85,B 0,C 180,E1 2298.383,E2 2298.383} C_VEL
LIN {X 0,Y 727.715,Z 749.56,A -85,B 0,C 180,E1 2302.101,E2 2302.101} C_VEL
LIN {X 0,Y 727.779,Z 749.56,A -85,B 0,C 180,E1 2306.156,E2 2306.156} C_VEL
LIN {X 0,Y 727.747,Z 749.56,A -85,B 0,C 180,E1 2310.706,E2 2310.706} C_VEL
LIN {X 0,Y 727.66,Z 749.56,A -85,B 0,C 180,E1 2315.455,E2 2315.455} C_VEL
LIN {X 0,Y 727.818,Z 749.56,A -85,B 0,C 180,E1 2320.594,E2 2320.594} C_VEL
LIN {X 0,Y 727.898,Z 749.56,A -85,B 0,C 180,E1 2325.571,E2 2325.571} C_VEL
LIN {X 0,Y 728.071,Z 749.56,A -85,B 0,C 180,E1 2330.439,E2 2330.439} C_VEL
LIN {X 0,Y 727.978,Z 749.56,A -85,B 0,C 180,E1 2335.234,E2 2335.234} C_VEL
LIN {X 0,Y 728.106,Z 749.56,A -85,B 0,C 180,E1 2339.997,E2 2339.997} C_VEL
LIN {X 0,Y 728.173,Z 749.56,A -85,B 0,C 180,E1 2345.048,E2 2345.048} C_VEL
LIN {X 0,Y 728.006,Z 749.56,A -85,B 0,C 180,E1 2346.246,E2 2346.246} C_VEL
LIN {X 0,Y 724.067,Z 749.56,A -85,B 0,C 180,E1 2347.588,E2 2347.588} C_VEL
LIN {X 0,Y 720.152,Z 749.56,A -85,B 0,C 180,E1 2348.944,E2 2348.944} C_VEL
LIN {X 0,Y 720.076,Z 749.56,A -85,B 0,C 180,E1 2353.344,E2 2353.344} C_VEL
LIN {X 0,Y 720.06,Z 749.56,A -85,B 0,C 180,E1 2358.345,E2 2358.345} C_VEL
LIN {X 0,Y 720.072,Z 749.56,A -85,B 0,C 180,E1 2363.496,E2 2363.496} C_VEL
LIN {X 0,Y 720.004,Z 749.56,A -85,B 0,C 180,E1 2368.86,E2 2368.86} C_VEL
LIN {X 0,Y 720.061,Z 749.56,A -85,B 0,C 180,E1 2373.065,E2 2373.065} C_VEL
LIN {X 0,Y 719.94,Z 749.56,A -85,B 0,C 180,E1 2377.492,E2 2377.492} C_VEL
LIN {X 0,Y 720.018,Z 749.56,A -85,B 0,C 180,E1 2382.729,E2 2382.729} C_VEL
LIN {X 0,Y 719.751,Z 749.56,A -85,B 0,C 180,E1 2387.289,E2 2387.289} C_VEL
LIN {X 0,Y 720.169,Z 749.56,A -85,B 0,C 180,E1 2390.926,E2 2390.926} C_VEL
LIN {X 0,Y 724.737,Z 759.676,A -85,B 0,C 180,E1 2391.361,E2 2391.361} C_VEL
LIN {X 0,Y 729.002,Z 769.149,A -85,B 0,C 180,E1 2391.745,E2 2391.745} C_VEL
LIN {X 0,Y 728.901,Z 847.08,A -85,B 0,C 180,E1 2392.806,E2 2392.806} C_VEL
LIN {X 0,Y 727.878,Z 891.684,A -85,B 0,C 180,E1 2393.834,E2 2393.834} C_VEL
LIN {X 0,Y 726.763,Z 939.016,A -85,B 0,C 180,E1 2395.453,E2 2395.453} C_VEL
LIN {X 0,Y 725.382,Z 987.011,A -85,B 0,C 180,E1 2397.671,E2 2397.671} C_VEL
LIN {X 0,Y 724.13,Z 1029.766,A -85,B 0,C 180,E1 2400.229,E2 2400.229} C_VEL
LIN {X 0,Y 722.956,Z 1069.003,A -85,B 0,C 180,E1 2403.134,E2 2403.134} C_VEL
LIN {X 0,Y 721.942,Z 1106.123,A -85,B 0,C 180,E1 2406.565,E2 2406.565} C_VEL
LIN {X 0,Y 721.206,Z 1135.572,A -85,B 0,C 180,E1 2409.933,E2 2409.933} C_VEL
LIN {X 0,Y 720.709,Z 1160.887,A -85,B 0,C 180,E1 2413.557,E2 2413.557} C_VEL
LIN {X 0,Y 720.473,Z 1180.016,A -85,B 0,C 180,E1 2417.063,E2 2417.063} C_VEL
LIN {X 0,Y 720.341,Z 1195.443,A -85,B 0,C 180,E1 2420.947,E2 2420.947} C_VEL
LIN {X 0,Y 720.259,Z 1204.797,A -85,B 0,C 180,E1 2424.582,E2 2424.582} C_VEL
LIN {X 0,Y 720.285,Z 1208.966,A -85,B 0,C 180,E1 2427.595,E2 2427.595} C_VEL
LIN {X 0,Y 720.438,Z 1209.669,A -85,B 0,C 180,E1 2431.201,E2 2431.201} C_VEL
LIN {X 0,Y 720.224,Z 1205.912,A -85,B 0,C 180,E1 2434.814,E2 2434.814} C_VEL
LIN {X 0,Y 720.173,Z 1197.334,A -85,B 0,C 180,E1 2438.446,E2 2438.446} C_VEL
LIN {X 0,Y 720.286,Z 1185.047,A -85,B 0,C 180,E1 2441.803,E2 2441.803} C_VEL
LIN {X 0,Y 720.544,Z 1167.791,A -85,B 0,C 180,E1 2445.274,E2 2445.274} C_VEL
LIN {X 0,Y 720.868,Z 1146.556,A -85,B 0,C 180,E1 2448.602,E2 2448.602} C_VEL
LIN {X 0,Y 721.553,Z 1119.829,A -85,B 0,C 180,E1 2451.96,E2 2451.96} C_VEL
LIN {X 0,Y 722.471,Z 1084.884,A -85,B 0,C 180,E1 2455.488,E2 2455.488} C_VEL
LIN {X 0,Y 723.557,Z 1047.015,A -85,B 0,C 180,E1 2458.567,E2 2458.567} C_VEL
LIN {X 0,Y 724.919,Z 1005.067,A -85,B 0,C 180,E1 2461.321,E2 2461.321} C_VEL
LIN {X 0,Y 726.27,Z 961.494,A -85,B 0,C 180,E1 2463.574,E2 2463.574} C_VEL
LIN {X 0,Y 727.487,Z 916.243,A -85,B 0,C 180,E1 2465.388,E2 2465.388} C_VEL
LIN {X 0,Y 728.416,Z 871.419,A -85,B 0,C 180,E1 2466.687,E2 2466.687} C_VEL
LIN {X 0,Y 729.039,Z 826.513,A -85,B 0,C 180,E1 2467.534,E2 2467.534} C_VEL
LIN {X 0,Y 728.415,Z 766.398,A -85,B 0,C 180,E1 2468.325,E2 2468.325} C_VEL
LIN {X 0,Y 719.947,Z 751.086,A -85,B 0,C 180,E1 2469.052,E2 2469.052} C_VEL
LIN {X 0,Y 719.783,Z 749.56,A -85,B 0,C 180,E1 2469.108,E2 2469.108} C_VEL
LIN {X 0,Y 720.077,Z 749.56,A -85,B 0,C 180,E1 2473.83,E2 2473.83} C_VEL
LIN {X 0,Y 719.864,Z 749.56,A -85,B 0,C 180,E1 2479.405,E2 2479.405} C_VEL
LIN {X 0,Y 719.855,Z 749.56,A -85,B 0,C 180,E1 2484.004,E2 2484.004} C_VEL
LIN {X 0,Y 719.876,Z 749.56,A -85,B 0,C 180,E1 2489.389,E2 2489.389} C_VEL
LIN {X 0,Y 719.904,Z 749.56,A -85,B 0,C 180,E1 2494.5,E2 2494.5} C_VEL
LIN {X 0,Y 719.927,Z 749.56,A -85,B 0,C 180,E1 2499.097,E2 2499.097} C_VEL
LIN {X 0,Y 720.145,Z 749.56,A -85,B 0,C 180,E1 2504.173,E2 2504.173} C_VEL
LIN {X 0,Y 720.059,Z 749.56,A -85,B 0,C 180,E1 2509.116,E2 2509.116} C_VEL
LIN {X 0,Y 720.128,Z 749.56,A -85,B 0,C 180,E1 2513.981,E2 2513.981} C_VEL
LIN {X 0,Y 720.374,Z 749.56,A -85,B 0,C 180,E1 2518.801,E2 2518.801} C_VEL
LIN {X 0,Y 720.246,Z 749.56,A -85,B 0,C 180,E1 2523.612,E2 2523.612} C_VEL
LIN {X 0,Y 720.06,Z 749.56,A -85,B 0,C 180,E1 2528.451,E2 2528.451} C_VEL
LIN {X 0,Y 719.957,Z 749.56,A -85,B 0,C 180,E1 2532.12,E2 2532.12} C_VEL
LIN {X 0,Y 719.794,Z 749.56,A -85,B 0,C 180,E1 2535.842,E2 2535.842} C_VEL
LIN {X 0,Y 719.935,Z 749.56,A -85,B 0,C 180,E1 2540.91,E2 2540.91} C_VEL
LIN {X 0,Y 719.889,Z 749.56,A -85,B 0,C 180,E1 2546.16,E2 2546.16} C_VEL
LIN {X 0,Y 719.843,Z 749.56,A -85,B 0,C 180,E1 2551.66,E2 2551.66} C_VEL
LIN {X 0,Y 719.829,Z 749.56,A -85,B 0,C 180,E1 2556.006,E2 2556.006} C_VEL
LIN {X 0,Y 719.821,Z 749.56,A -85,B 0,C 180,E1 2560.91,E2 2560.91} C_VEL
LIN {X 0,Y 720.088,Z 749.762,A -85,B 0,C 180,E1 2566.218,E2 2566.218} C_VEL
LIN {X 0,Y 727.323,Z 765.686,A -85,B 0,C 180,E1 2566.799,E2 2566.799} C_VEL
LIN {X 0,Y 726.973,Z 815.143,A -85,B 0,C 180,E1 2567.62,E2 2567.62} C_VEL
LIN {X 0,Y 726.272,Z 861.191,A -85,B 0,C 180,E1 2568.887,E2 2568.887} C_VEL
LIN {X 0,Y 725.045,Z 907.843,A -85,B 0,C 180,E1 2570.73,E2 2570.73} C_VEL
LIN {X 0,Y 723.976,Z 949.518,A -85,B 0,C 180,E1 2572.929,E2 2572.929} C_VEL
LIN {X 0,Y 722.871,Z 988.761,A -85,B 0,C 180,E1 2575.556,E2 2575.556} C_VEL
LIN {X 0,Y 721.913,Z 1026.347,A -85,B 0,C 180,E1 2578.747,E2 2578.747} C_VEL
LIN {X 0,Y 721.111,Z 1057.413,A -85,B 0,C 180,E1 2582.092,E2 2582.092} C_VEL
LIN {X 0,Y 720.63,Z 1081.964,A -85,B 0,C 180,E1 2585.45,E2 2585.45} C_VEL
LIN {X 0,Y 720.501,Z 1100.841,A -85,B 0,C 180,E1 2588.789,E2 2588.789} C_VEL
LIN {X 0,Y 720.31,Z 1114.708,A -85,B 0,C 180,E1 2592.086,E2 2592.086} C_VEL
LIN {X 0,Y 720.31,Z 1124.014,A -85,B 0,C 180,E1 2595.42,E2 2595.42} C_VEL
LIN {X 0,Y 720.177,Z 1129.277,A -85,B 0,C 180,E1 2599.115,E2 2599.115} C_VEL
LIN {X 0,Y 720.373,Z 1129.297,A -85,B 0,C 180,E1 2602.77,E2 2602.77} C_VEL
LIN {X 0,Y 720.393,Z 1124.208,A -85,B 0,C 180,E1 2606.393,E2 2606.393} C_VEL
LIN {X 0,Y 720.424,Z 1114.041,A -85,B 0,C 180,E1 2610.001,E2 2610.001} C_VEL
LIN {X 0,Y 720.534,Z 1096.882,A -85,B 0,C 180,E1 2613.909,E2 2613.909} C_VEL
LIN {X 0,Y 720.875,Z 1074.758,A -85,B 0,C 180,E1 2617.529,E2 2617.529} C_VEL
LIN {X 0,Y 721.357,Z 1048.462,A -85,B 0,C 180,E1 2620.868,E2 2620.868} C_VEL
LIN {X 0,Y 722.218,Z 1014.714,A -85,B 0,C 180,E1 2624.233,E2 2624.233} C_VEL
LIN {X 0,Y 723.215,Z 976.361,A -85,B 0,C 180,E1 2627.25,E2 2627.25} C_VEL
LIN {X 0,Y 724.298,Z 937.437,A -85,B 0,C 180,E1 2629.675,E2 2629.675} C_VEL
LIN {X 0,Y 725.508,Z 895.241,A -85,B 0,C 180,E1 2631.736,E2 2631.736} C_VEL
LIN {X 0,Y 726.496,Z 849.901,A -85,B 0,C 180,E1 2633.376,E2 2633.376} C_VEL
LIN {X 0,Y 727.285,Z 804.004,A -85,B 0,C 180,E1 2634.518,E2 2634.518} C_VEL
LIN {X 0,Y 727.031,Z 765.283,A -85,B 0,C 180,E1 2635.131,E2 2635.131} C_VEL
LIN {X 0,Y 719.882,Z 749.56,A -85,B 0,C 180,E1 2635.742,E2 2635.742} C_VEL
LIN {X 0,Y 719.87,Z 749.56,A -85,B 0,C 180,E1 2640.601,E2 2640.601} C_VEL
LIN {X 0,Y 719.826,Z 749.56,A -85,B 0,C 180,E1 2645.035,E2 2645.035} C_VEL
LIN {X 0,Y 719.765,Z 749.56,A -85,B 0,C 180,E1 2649.039,E2 2649.039} C_VEL
LIN {X 0,Y 720.06,Z 749.56,A -85,B 0,C 180,E1 2653.833,E2 2653.833} C_VEL
LIN {X 0,Y 719.879,Z 749.56,A -85,B 0,C 180,E1 2659.398,E2 2659.398} C_VEL
LIN {X 0,Y 719.821,Z 749.56,A -85,B 0,C 180,E1 2664.959,E2 2664.959} C_VEL
LIN {X 0,Y 719.842,Z 749.56,A -85,B 0,C 180,E1 2669.742,E2 2669.742} C_VEL
LIN {X 0,Y 719.861,Z 749.56,A -85,B 0,C 180,E1 2674.51,E2 2674.51} C_VEL
LIN {X 0,Y 719.908,Z 749.56,A -85,B 0,C 180,E1 2680.372,E2 2680.372} C_VEL
LIN {X 0,Y 719.956,Z 749.56,A -85,B 0,C 180,E1 2685.408,E2 2685.408} C_VEL
LIN {X 0,Y 720.171,Z 749.56,A -85,B 0,C 180,E1 2690.472,E2 2690.472} C_VEL
LIN {X 0,Y 720.111,Z 749.56,A -85,B 0,C 180,E1 2695.182,E2 2695.182} C_VEL
LIN {X 0,Y 720.224,Z 749.56,A -85,B 0,C 180,E1 2699.997,E2 2699.997} C_VEL
LIN {X 0,Y 720.347,Z 749.56,A -85,B 0,C 180,E1 2704.81,E2 2704.81} C_VEL
LIN {X 0,Y 720.152,Z 749.56,A -85,B 0,C 180,E1 2708.944,E2 2708.944} C_VEL
LIN {X 0,Y 716.113,Z 749.56,A -85,B 0,C 180,E1 2710.298,E2 2710.298} C_VEL
LIN {X 0,Y 712.141,Z 749.56,A -85,B 0,C 180,E1 2711.668,E2 2711.668} C_VEL
LIN {X 0,Y 712.266,Z 749.56,A -85,B 0,C 180,E1 2717.308,E2 2717.308} C_VEL
LIN {X 0,Y 712.095,Z 749.56,A -85,B 0,C 180,E1 2722.453,E2 2722.453} C_VEL
LIN {X 0,Y 712.045,Z 749.56,A -85,B 0,C 180,E1 2726.957,E2 2726.957} C_VEL
LIN {X 0,Y 712.096,Z 749.56,A -85,B 0,C 180,E1 2732.038,E2 2732.038} C_VEL
LIN {X 0,Y 712.032,Z 749.56,A -85,B 0,C 180,E1 2736.455,E2 2736.455} C_VEL
LIN {X 0,Y 712.056,Z 749.56,A -85,B 0,C 180,E1 2742.031,E2 2742.031} C_VEL
LIN {X 0,Y 711.963,Z 749.56,A -85,B 0,C 180,E1 2746.187,E2 2746.187} C_VEL
LIN {X 0,Y 712.131,Z 749.803,A -85,B 0,C 180,E1 2750.419,E2 2750.419} C_VEL
LIN {X 0,Y 717.028,Z 759.913,A -85,B 0,C 180,E1 2750.87,E2 2750.87} C_VEL
LIN {X 0,Y 722.805,Z 770.866,A -85,B 0,C 180,E1 2751.378,E2 2751.378} C_VEL
LIN {X 0,Y 722.602,Z 847.183,A -85,B 0,C 180,E1 2752.428,E2 2752.428} C_VEL
LIN {X 0,Y 721.435,Z 891.194,A -85,B 0,C 180,E1 2753.445,E2 2753.445} C_VEL
LIN {X 0,Y 720.158,Z 938.152,A -85,B 0,C 180,E1 2755.054,E2 2755.054} C_VEL
LIN {X 0,Y 718.481,Z 986.088,A -85,B 0,C 180,E1 2757.273,E2 2757.273} C_VEL
LIN {X 0,Y 717.08,Z 1027.751,A -85,B 0,C 180,E1 2759.765,E2 2759.765} C_VEL
LIN {X 0,Y 715.642,Z 1068.135,A -85,B 0,C 180,E1 2762.766,E2 2762.766} C_VEL
LIN {X 0,Y 714.391,Z 1103.94,A -85,B 0,C 180,E1 2766.078,E2 2766.078} C_VEL
LIN {X 0,Y 713.575,Z 1134.356,A -85,B 0,C 180,E1 2769.548,E2 2769.548} C_VEL
LIN {X 0,Y 712.947,Z 1160.889,A -85,B 0,C 180,E1 2773.372,E2 2773.372} C_VEL
LIN {X 0,Y 712.62,Z 1180.215,A -85,B 0,C 180,E1 2776.959,E2 2776.959} C_VEL
LIN {X 0,Y 712.475,Z 1195.652,A -85,B 0,C 180,E1 2780.912,E2 2780.912} C_VEL
LIN {X 0,Y 712.366,Z 1204.797,A -85,B 0,C 180,E1 2784.522,E2 2784.522} C_VEL
LIN {X 0,Y 712.383,Z 1208.963,A -85,B 0,C 180,E1 2787.568,E2 2787.568} C_VEL
LIN {X 0,Y 712.536,Z 1209.669,A -85,B 0,C 180,E1 2791.215,E2 2791.215} C_VEL
LIN {X 0,Y 712.332,Z 1205.912,A -85,B 0,C 180,E1 2794.867,E2 2794.867} C_VEL
LIN {X 0,Y 712.289,Z 1197.334,A -85,B 0,C 180,E1 2798.54,E2 2798.54} C_VEL
LIN {X 0,Y 712.4,Z 1185.049,A -85,B 0,C 180,E1 2801.935,E2 2801.935} C_VEL
LIN {X 0,Y 712.715,Z 1167.792,A -85,B 0,C 180,E1 2805.446,E2 2805.446} C_VEL
LIN {X 0,Y 713.105,Z 1146.735,A -85,B 0,C 180,E1 2808.787,E2 2808.787} C_VEL
LIN {X 0,Y 713.881,Z 1119.471,A -85,B 0,C 180,E1 2812.249,E2 2812.249} C_VEL
LIN {X 0,Y 715.005,Z 1084.281,A -85,B 0,C 180,E1 2815.832,E2 2815.832} C_VEL
LIN {X 0,Y 716.3,Z 1047.016,A -85,B 0,C 180,E1 2818.883,E2 2818.883} C_VEL
LIN {X 0,Y 717.883,Z 1005.822,A -85,B 0,C 180,E1 2821.62,E2 2821.62} C_VEL
LIN {X 0,Y 719.468,Z 961.498,A -85,B 0,C 180,E1 2823.935,E2 2823.935} C_VEL
LIN {X 0,Y 720.893,Z 917.115,A -85,B 0,C 180,E1 2825.727,E2 2825.727} C_VEL
LIN {X 0,Y 722.005,Z 871.886,A -85,B 0,C 180,E1 2827.055,E2 2827.055} C_VEL
LIN {X 0,Y 722.764,Z 826.481,A -85,B 0,C 180,E1 2827.918,E2 2827.918} C_VEL
LIN {X 0,Y 722.518,Z 770.124,A -85,B 0,C 180,E1 2828.649,E2 2828.649} C_VEL
LIN {X 0,Y 712.042,Z 751.199,A -85,B 0,C 180,E1 2829.569,E2 2829.569} C_VEL
LIN {X 0,Y 711.858,Z 749.56,A -85,B 0,C 180,E1 2829.654,E2 2829.654} C_VEL
LIN {X 0,Y 712.176,Z 749.56,A -85,B 0,C 180,E1 2834.443,E2 2834.443} C_VEL
LIN {X 0,Y 711.963,Z 749.56,A -85,B 0,C 180,E1 2840.454,E2 2840.454} C_VEL
LIN {X 0,Y 711.89,Z 749.56,A -85,B 0,C 180,E1 2845.878,E2 2845.878} C_VEL
LIN {X 0,Y 711.891,Z 749.56,A -85,B 0,C 180,E1 2850.779,E2 2850.779} C_VEL
LIN {X 0,Y 711.913,Z 749.56,A -85,B 0,C 180,E1 2855.884,E2 2855.884} C_VEL
LIN {X 0,Y 711.975,Z 749.56,A -85,B 0,C 180,E1 2860.151,E2 2860.151} C_VEL
LIN {X 0,Y 712.219,Z 749.56,A -85,B 0,C 180,E1 2863.992,E2 2863.992} C_VEL
LIN {X 0,Y 712.153,Z 749.56,A -85,B 0,C 180,E1 2868.994,E2 2868.994} C_VEL
LIN {X 0,Y 712.249,Z 749.56,A -85,B 0,C 180,E1 2873.914,E2 2873.914} C_VEL
LIN {X 0,Y 712.468,Z 749.56,A -85,B 0,C 180,E1 2878.788,E2 2878.788} C_VEL
LIN {X 0,Y 712.25,Z 749.56,A -85,B 0,C 180,E1 2884.325,E2 2884.325} C_VEL
LIN {X 0,Y 712.16,Z 749.56,A -85,B 0,C 180,E1 2888.546,E2 2888.546} C_VEL
LIN {X 0,Y 712.027,Z 749.56,A -85,B 0,C 180,E1 2892.514,E2 2892.514} C_VEL
LIN {X 0,Y 711.765,Z 749.56,A -85,B 0,C 180,E1 2897.295,E2 2897.295} C_VEL
LIN {X 0,Y 711.979,Z 749.56,A -85,B 0,C 180,E1 2901.154,E2 2901.154} C_VEL
LIN {X 0,Y 711.914,Z 749.56,A -85,B 0,C 180,E1 2906.939,E2 2906.939} C_VEL
LIN {X 0,Y 711.91,Z 749.56,A -85,B 0,C 180,E1 2912.055,E2 2912.055} C_VEL
LIN {X 0,Y 711.899,Z 749.56,A -85,B 0,C 180,E1 2916.471,E2 2916.471} C_VEL
LIN {X 0,Y 711.878,Z 749.56,A -85,B 0,C 180,E1 2921.157,E2 2921.157} C_VEL
LIN {X 0,Y 712.167,Z 749.56,A -85,B 0,C 180,E1 2925.762,E2 2925.762} C_VEL
LIN {X 0,Y 720.855,Z 768.313,A -85,B 0,C 180,E1 2926.481,E2 2926.481} C_VEL
LIN {X 0,Y 720.301,Z 818.355,A -85,B 0,C 180,E1 2927.344,E2 2927.344} C_VEL
LIN {X 0,Y 719.411,Z 863.465,A -85,B 0,C 180,E1 2928.627,E2 2928.627} C_VEL
LIN {X 0,Y 718.003,Z 909.728,A -85,B 0,C 180,E1 2930.49,E2 2930.49} C_VEL
LIN {X 0,Y 716.648,Z 952.494,A -85,B 0,C 180,E1 2932.802,E2 2932.802} C_VEL
LIN {X 0,Y 715.398,Z 990.492,A -85,B 0,C 180,E1 2935.41,E2 2935.41} C_VEL
LIN {X 0,Y 714.325,Z 1025.667,A -85,B 0,C 180,E1 2938.432,E2 2938.432} C_VEL
LIN {X 0,Y 713.457,Z 1056.78,A -85,B 0,C 180,E1 2941.806,E2 2941.806} C_VEL
LIN {X 0,Y 712.947,Z 1081.129,A -85,B 0,C 180,E1 2945.144,E2 2945.144} C_VEL
LIN {X 0,Y 712.603,Z 1102.209,A -85,B 0,C 180,E1 2948.929,E2 2948.929} C_VEL
LIN {X 0,Y 712.409,Z 1115.246,A -85,B 0,C 180,E1 2952.152,E2 2952.152} C_VEL
LIN {X 0,Y 712.391,Z 1125.046,A -85,B 0,C 180,E1 2955.882,E2 2955.882} C_VEL
LIN {X 0,Y 712.268,Z 1129.192,A -85,B 0,C 180,E1 2958.993,E2 2958.993} C_VEL
LIN {X 0,Y 712.459,Z 1129.382,A -85,B 0,C 180,E1 2962.689,E2 2962.689} C_VEL
LIN {X 0,Y 712.489,Z 1124.407,A -85,B 0,C 180,E1 2966.353,E2 2966.353} C_VEL
LIN {X 0,Y 712.529,Z 1114.417,A -85,B 0,C 180,E1 2970.001,E2 2970.001} C_VEL
LIN {X 0,Y 712.761,Z 1098.895,A -85,B 0,C 180,E1 2973.647,E2 2973.647} C_VEL
LIN {X 0,Y 713.086,Z 1077.589,A -85,B 0,C 180,E1 2977.305,E2 2977.305} C_VEL
LIN {X 0,Y 713.655,Z 1049.394,A -85,B 0,C 180,E1 2980.987,E2 2980.987} C_VEL
LIN {X 0,Y 714.622,Z 1015.862,A -85,B 0,C 180,E1 2984.387,E2 2984.387} C_VEL
LIN {X 0,Y 715.795,Z 979.276,A -85,B 0,C 180,E1 2987.329,E2 2987.329} C_VEL
LIN {X 0,Y 717.098,Z 940.404,A -85,B 0,C 180,E1 2989.822,E2 2989.822} C_VEL
LIN {X 0,Y 718.496,Z 897.094,A -85,B 0,C 180,E1 2991.984,E2 2991.984} C_VEL
LIN {X 0,Y 719.644,Z 853.35,A -85,B 0,C 180,E1 2993.612,E2 2993.612} C_VEL
LIN {X 0,Y 720.664,Z 806.007,A -85,B 0,C 180,E1 2994.83,E2 2994.83} C_VEL
LIN {X 0,Y 720.563,Z 768.138,A -85,B 0,C 180,E1 2995.447,E2 2995.447} C_VEL
LIN {X 0,Y 711.957,Z 749.56,A -85,B 0,C 180,E1 2996.187,E2 2996.187} C_VEL
LIN {X 0,Y 711.972,Z 749.56,A -85,B 0,C 180,E1 3000.624,E2 3000.624} C_VEL
LIN {X 0,Y 711.933,Z 749.56,A -85,B 0,C 180,E1 3004.967,E2 3004.967} C_VEL
LIN {X 0,Y 711.816,Z 749.56,A -85,B 0,C 180,E1 3010.153,E2 3010.153} C_VEL
LIN {X 0,Y 712.149,Z 749.56,A -85,B 0,C 180,E1 3014.447,E2 3014.447} C_VEL
LIN {X 0,Y 711.996,Z 749.56,A -85,B 0,C 180,E1 3020.447,E2 3020.447} C_VEL
LIN {X 0,Y 711.882,Z 749.56,A -85,B 0,C 180,E1 3025.881,E2 3025.881} C_VEL
LIN {X 0,Y 711.862,Z 749.56,A -85,B 0,C 180,E1 3030.77,E2 3030.77} C_VEL
LIN {X 0,Y 711.894,Z 749.56,A -85,B 0,C 180,E1 3034.874,E2 3034.874} C_VEL
LIN {X 0,Y 711.98,Z 749.56,A -85,B 0,C 180,E1 3040.144,E2 3040.144} C_VEL
LIN {X 0,Y 712.046,Z 749.56,A -85,B 0,C 180,E1 3045.242,E2 3045.242} C_VEL
LIN {X 0,Y 712.278,Z 749.56,A -85,B 0,C 180,E1 3050.225,E2 3050.225} C_VEL
LIN {X 0,Y 712.22,Z 749.56,A -85,B 0,C 180,E1 3055.128,E2 3055.128} C_VEL
LIN {X 0,Y 712.323,Z 749.56,A -85,B 0,C 180,E1 3059.997,E2 3059.997} C_VEL
LIN {X 0,Y 712.446,Z 749.56,A -85,B 0,C 180,E1 3064.864,E2 3064.864} C_VEL
LIN {X 0,Y 712.192,Z 749.56,A -85,B 0,C 180,E1 3069.77,E2 3069.77} C_VEL
LIN {X 0,Y 712.141,Z 749.56,A -85,B 0,C 180,E1 3071.668,E2 3071.668} C_VEL
LIN {X 0,Y 710.906,Z 749.56,A -85,B 0,C 180,E1 3072.363,E2 3072.363} C_VEL
LIN {X 0,Y 704.294,Z 749.56,A -85,B 0,C 180,E1 3074.25,E2 3074.25} C_VEL
LIN {X 0,Y 704.205,Z 749.56,A -85,B 0,C 180,E1 3074.429,E2 3074.429} C_VEL
LIN {X 0,Y 704.278,Z 749.56,A -85,B 0,C 180,E1 3079.25,E2 3079.25} C_VEL
LIN {X 0,Y 704.231,Z 749.56,A -85,B 0,C 180,E1 3084.057,E2 3084.057} C_VEL
LIN {X 0,Y 704.121,Z 749.56,A -85,B 0,C 180,E1 3089.575,E2 3089.575} C_VEL
LIN {X 0,Y 704.139,Z 749.56,A -85,B 0,C 180,E1 3093.913,E2 3093.913} C_VEL
LIN {X 0,Y 703.961,Z 749.56,A -85,B 0,C 180,E1 3098.497,E2 3098.497} C_VEL
LIN {X 0,Y 704.235,Z 749.56,A -85,B 0,C 180,E1 3103.362,E2 3103.362} C_VEL
LIN {X 0,Y 703.992,Z 749.56,A -85,B 0,C 180,E1 3108.698,E2 3108.698} C_VEL
LIN {X 0,Y 704.133,Z 749.857,A -85,B 0,C 180,E1 3109.88,E2 3109.88} C_VEL
LIN {X 0,Y 709.209,Z 760.11,A -85,B 0,C 180,E1 3110.357,E2 3110.357} C_VEL
LIN {X 0,Y 716.693,Z 773.972,A -85,B 0,C 180,E1 3111.026,E2 3111.026} C_VEL
LIN {X 0,Y 716.339,Z 846.816,A -85,B 0,C 180,E1 3112.035,E2 3112.035} C_VEL
LIN {X 0,Y 715.025,Z 890.508,A -85,B 0,C 180,E1 3113.042,E2 3113.042} C_VEL
LIN {X 0,Y 713.519,Z 938.371,A -85,B 0,C 180,E1 3114.69,E2 3114.69} C_VEL
LIN {X 0,Y 711.608,Z 986.091,A -85,B 0,C 180,E1 3116.916,E2 3116.916} C_VEL
LIN {X 0,Y 709.898,Z 1028.939,A -85,B 0,C 180,E1 3119.511,E2 3119.511} C_VEL
LIN {X 0,Y 708.221,Z 1069.41,A -85,B 0,C 180,E1 3122.564,E2 3122.564} C_VEL
LIN {X 0,Y 706.729,Z 1107.3,A -85,B 0,C 180,E1 3126.153,E2 3126.153} C_VEL
LIN {X 0,Y 705.722,Z 1138.012,A -85,B 0,C 180,E1 3129.801,E2 3129.801} C_VEL
LIN {X 0,Y 705.066,Z 1162.846,A -85,B 0,C 180,E1 3133.502,E2 3133.502} C_VEL
LIN {X 0,Y 704.69,Z 1181.694,A -85,B 0,C 180,E1 3137.151,E2 3137.151} C_VEL
LIN {X 0,Y 704.574,Z 1196.134,A -85,B 0,C 180,E1 3140.966,E2 3140.966} C_VEL
LIN {X 0,Y 704.483,Z 1204.797,A -85,B 0,C 180,E1 3144.46,E2 3144.46} C_VEL
LIN {X 0,Y 704.498,Z 1208.96,A -85,B 0,C 180,E1 3147.541,E2 3147.541} C_VEL
LIN {X 0,Y 704.633,Z 1209.669,A -85,B 0,C 180,E1 3151.228,E2 3151.228} C_VEL
LIN {X 0,Y 704.428,Z 1205.912,A -85,B 0,C 180,E1 3154.922,E2 3154.922} C_VEL
LIN {X 0,Y 704.412,Z 1197.334,A -85,B 0,C 180,E1 3158.636,E2 3158.636} C_VEL
LIN {X 0,Y 704.536,Z 1185.05,A -85,B 0,C 180,E1 3162.07,E2 3162.07} C_VEL
LIN {X 0,Y 704.888,Z 1167.503,A -85,B 0,C 180,E1 3165.674,E2 3165.674} C_VEL
LIN {X 0,Y 705.495,Z 1144.399,A -85,B 0,C 180,E1 3169.342,E2 3169.342} C_VEL
LIN {X 0,Y 706.349,Z 1115.095,A -85,B 0,C 180,E1 3172.994,E2 3172.994} C_VEL
LIN {X 0,Y 707.648,Z 1081.51,A -85,B 0,C 180,E1 3176.378,E2 3176.378} C_VEL
LIN {X 0,Y 709.347,Z 1041.608,A -85,B 0,C 180,E1 3179.607,E2 3179.607} C_VEL
LIN {X 0,Y 711.067,Z 1000.142,A -85,B 0,C 180,E1 3182.295,E2 3182.295} C_VEL
LIN {X 0,Y 712.992,Z 955.32,A -85,B 0,C 180,E1 3184.586,E2 3184.586} C_VEL
LIN {X 0,Y 714.52,Z 912.715,A -85,B 0,C 180,E1 3186.254,E2 3186.254} C_VEL
LIN {X 0,Y 715.678,Z 870.878,A -85,B 0,C 180,E1 3187.464,E2 3187.464} C_VEL
LIN {X 0,Y 716.566,Z 823.959,A -85,B 0,C 180,E1 3188.342,E2 3188.342} C_VEL
LIN {X 0,Y 716.05,Z 772.934,A -85,B 0,C 180,E1 3189.029,E2 3189.029} C_VEL
LIN {X 0,Y 704.159,Z 751.393,A -85,B 0,C 180,E1 3190.099,E2 3190.099} C_VEL
LIN {X 0,Y 703.941,Z 749.56,A -85,B 0,C 180,E1 3190.244,E2 3190.244} C_VEL
LIN {X 0,Y 704.217,Z 749.56,A -85,B 0,C 180,E1 3195.082,E2 3195.082} C_VEL
LIN {X 0,Y 704.043,Z 749.56,A -85,B 0,C 180,E1 3200.595,E2 3200.595} C_VEL
LIN {X 0,Y 703.981,Z 749.56,A -85,B 0,C 180,E1 3206.079,E2 3206.079} C_VEL
LIN {X 0,Y 704.014,Z 749.56,A -85,B 0,C 180,E1 3210.42,E2 3210.42} C_VEL
LIN {X 0,Y 704.055,Z 749.56,A -85,B 0,C 180,E1 3214.582,E2 3214.582} C_VEL
LIN {X 0,Y 704.063,Z 749.56,A -85,B 0,C 180,E1 3219.919,E2 3219.919} C_VEL
LIN {X 0,Y 704.236,Z 749.56,A -85,B 0,C 180,E1 3224.925,E2 3224.925} C_VEL
LIN {X 0,Y 704.295,Z 749.56,A -85,B 0,C 180,E1 3230.12,E2 3230.12} C_VEL
LIN {X 0,Y 704.53,Z 749.56,A -85,B 0,C 180,E1 3235.082,E2 3235.082} C_VEL
LIN {X 0,Y 704.394,Z 749.56,A -85,B 0,C 180,E1 3240.003,E2 3240.003} C_VEL
LIN {X 0,Y 704.32,Z 749.56,A -85,B 0,C 180,E1 3244.927,E2 3244.927} C_VEL
LIN {X 0,Y 704.369,Z 749.56,A -85,B 0,C 180,E1 3249.886,E2 3249.886} C_VEL
LIN {X 0,Y 704.076,Z 749.56,A -85,B 0,C 180,E1 3255.027,E2 3255.027} C_VEL
LIN {X 0,Y 704.07,Z 749.56,A -85,B 0,C 180,E1 3260.089,E2 3260.089} C_VEL
LIN {X 0,Y 703.946,Z 749.56,A -85,B 0,C 180,E1 3265.633,E2 3265.633} C_VEL
LIN {X 0,Y 704.023,Z 749.56,A -85,B 0,C 180,E1 3271.012,E2 3271.012} C_VEL
LIN {X 0,Y 704.005,Z 749.56,A -85,B 0,C 180,E1 3275.424,E2 3275.424} C_VEL
LIN {X 0,Y 704.043,Z 749.56,A -85,B 0,C 180,E1 3280.089,E2 3280.089} C_VEL
LIN {X 0,Y 704.275,Z 750.358,A -85,B 0,C 180,E1 3285.329,E2 3285.329} C_VEL
LIN {X 0,Y 714.375,Z 772.949,A -85,B 0,C 180,E1 3286.186,E2 3286.186} C_VEL
LIN {X 0,Y 713.673,Z 822.748,A -85,B 0,C 180,E1 3287.092,E2 3287.092} C_VEL
LIN {X 0,Y 712.492,Z 868.585,A -85,B 0,C 180,E1 3288.464,E2 3288.464} C_VEL
LIN {X 0,Y 710.916,Z 912.617,A -85,B 0,C 180,E1 3290.297,E2 3290.297} C_VEL
LIN {X 0,Y 709.317,Z 956.611,A -85,B 0,C 180,E1 3292.744,E2 3292.744} C_VEL
LIN {X 0,Y 707.845,Z 994.614,A -85,B 0,C 180,E1 3295.451,E2 3295.451} C_VEL
LIN {X 0,Y 706.647,Z 1028.526,A -85,B 0,C 180,E1 3298.465,E2 3298.465} C_VEL
LIN {X 0,Y 705.661,Z 1059.296,A -85,B 0,C 180,E1 3301.894,E2 3301.894} C_VEL
LIN {X 0,Y 704.989,Z 1084.203,A -85,B 0,C 180,E1 3305.459,E2 3305.459} C_VEL
LIN {X 0,Y 704.722,Z 1103.128,A -85,B 0,C 180,E1 3308.985,E2 3308.985} C_VEL
LIN {X 0,Y 704.468,Z 1116.713,A -85,B 0,C 180,E1 3312.525,E2 3312.525} C_VEL
LIN {X 0,Y 704.49,Z 1124.843,A -85,B 0,C 180,E1 3315.72,E2 3315.72} C_VEL
LIN {X 0,Y 704.358,Z 1129.107,A -85,B 0,C 180,E1 3318.868,E2 3318.868} C_VEL
LIN {X 0,Y 704.545,Z 1129.466,A -85,B 0,C 180,E1 3322.607,E2 3322.607} C_VEL
LIN {X 0,Y 704.585,Z 1124.605,A -85,B 0,C 180,E1 3326.312,E2 3326.312} C_VEL
LIN {X 0,Y 704.635,Z 1114.787,A -85,B 0,C 180,E1 3330.001,E2 3330.001} C_VEL
LIN {X 0,Y 704.888,Z 1099.403,A -85,B 0,C 180,E1 3333.688,E2 3333.688} C_VEL
LIN {X 0,Y 705.262,Z 1078.299,A -85,B 0,C 180,E1 3337.387,E2 3337.387} C_VEL
LIN {X 0,Y 705.952,Z 1050.273,A -85,B 0,C 180,E1 3341.108,E2 3341.108} C_VEL
LIN {X 0,Y 707.016,Z 1018.675,A -85,B 0,C 180,E1 3344.387,E2 3344.387} C_VEL
LIN {X 0,Y 708.293,Z 983.706,A -85,B 0,C 180,E1 3347.299,E2 3347.299} C_VEL
LIN {X 0,Y 709.849,Z 944.336,A -85,B 0,C 180,E1 3349.915,E2 3349.915} C_VEL
LIN {X 0,Y 711.385,Z 901.267,A -85,B 0,C 180,E1 3352.133,E2 3352.133} C_VEL
LIN {X 0,Y 712.813,Z 857.272,A -85,B 0,C 180,E1 3353.837,E2 3353.837} C_VEL
LIN {X 0,Y 713.935,Z 809.401,A -85,B 0,C 180,E1 3355.115,E2 3355.115} C_VEL
LIN {X 0,Y 714.007,Z 770.821,A -85,B 0,C 180,E1 3355.774,E2 3355.774} C_VEL
LIN {X 0,Y 704.214,Z 751.227,A -85,B 0,C 180,E1 3356.574,E2 3356.574} C_VEL
LIN {X 0,Y 704.061,Z 749.56,A -85,B 0,C 180,E1 3356.642,E2 3356.642} C_VEL
LIN {X 0,Y 704.06,Z 749.56,A -85,B 0,C 180,E1 3361.006,E2 3361.006} C_VEL
LIN {X 0,Y 704.03,Z 749.56,A -85,B 0,C 180,E1 3365.418,E2 3365.418} C_VEL
LIN {X 0,Y 703.915,Z 749.56,A -85,B 0,C 180,E1 3370.093,E2 3370.093} C_VEL
LIN {X 0,Y 704.175,Z 749.56,A -85,B 0,C 180,E1 3374.908,E2 3374.908} C_VEL
LIN {X 0,Y 704.072,Z 749.56,A -85,B 0,C 180,E1 3380.594,E2 3380.594} C_VEL
LIN {X 0,Y 703.976,Z 749.56,A -85,B 0,C 180,E1 3386.07,E2 3386.07} C_VEL
LIN {X 0,Y 703.98,Z 749.56,A -85,B 0,C 180,E1 3390.411,E2 3390.411} C_VEL
LIN {X 0,Y 703.974,Z 749.56,A -85,B 0,C 180,E1 3394.572,E2 3394.572} C_VEL
LIN {X 0,Y 704.06,Z 749.56,A -85,B 0,C 180,E1 3399.911,E2 3399.911} C_VEL
LIN {X 0,Y 704.101,Z 749.56,A -85,B 0,C 180,E1 3405.072,E2 3405.072} C_VEL
LIN {X 0,Y 704.377,Z 749.56,A -85,B 0,C 180,E1 3410.114,E2 3410.114} C_VEL
LIN {X 0,Y 704.319,Z 749.56,A -85,B 0,C 180,E1 3415.073,E2 3415.073} C_VEL
LIN {X 0,Y 704.423,Z 749.56,A -85,B 0,C 180,E1 3419.997,E2 3419.997} C_VEL
LIN {X 0,Y 704.53,Z 749.56,A -85,B 0,C 180,E1 3424.918,E2 3424.918} C_VEL
LIN {X 0,Y 704.301,Z 749.56,A -85,B 0,C 180,E1 3429.88,E2 3429.88} C_VEL
LIN {X 0,Y 704.205,Z 749.56,A -85,B 0,C 180,E1 3434.429,E2 3434.429} C_VEL
LIN {X 0,Y 700.292,Z 749.56,A -85,B 0,C 180,E1 3435.819,E2 3435.819} C_VEL
LIN {X 0,Y 696.428,Z 749.56,A -85,B 0,C 180,E1 3437.225,E2 3437.225} C_VEL
LIN {X 0,Y 696.297,Z 749.56,A -85,B 0,C 180,E1 3441.647,E2 3441.647} C_VEL
LIN {X 0,Y 696.295,Z 749.56,A -85,B 0,C 180,E1 3445.722,E2 3445.722} C_VEL
LIN {X 0,Y 696.183,Z 749.56,A -85,B 0,C 180,E1 3449.946,E2 3449.946} C_VEL
LIN {X 0,Y 696.162,Z 749.56,A -85,B 0,C 180,E1 3454.426,E2 3454.426} C_VEL
LIN {X 0,Y 696.019,Z 749.56,A -85,B 0,C 180,E1 3459.019,E2 3459.019} C_VEL
LIN {X 0,Y 696.271,Z 749.56,A -85,B 0,C 180,E1 3464.257,E2 3464.257} C_VEL
LIN {X 0,Y 696.139,Z 749.878,A -85,B 0,C 180,E1 3469.323,E2 3469.323} C_VEL
LIN {X 0,Y 701.365,Z 760.271,A -85,B 0,C 180,E1 3469.826,E2 3469.826} C_VEL
LIN {X 0,Y 710.566,Z 776.958,A -85,B 0,C 180,E1 3470.663,E2 3470.663} C_VEL
LIN {X 0,Y 710.029,Z 848.606,A -85,B 0,C 180,E1 3471.672,E2 3471.672} C_VEL
LIN {X 0,Y 708.598,Z 892.435,A -85,B 0,C 180,E1 3472.709,E2 3472.709} C_VEL
LIN {X 0,Y 706.851,Z 939.966,A -85,B 0,C 180,E1 3474.377,E2 3474.377} C_VEL
LIN {X 0,Y 704.688,Z 988.043,A -85,B 0,C 180,E1 3476.656,E2 3476.656} C_VEL
LIN {X 0,Y 702.672,Z 1031.361,A -85,B 0,C 180,E1 3479.337,E2 3479.337} C_VEL
LIN {X 0,Y 700.869,Z 1069.489,A -85,B 0,C 180,E1 3482.259,E2 3482.259} C_VEL
LIN {X 0,Y 699.171,Z 1107.166,A -85,B 0,C 180,E1 3485.865,E2 3485.865} C_VEL
LIN {X 0,Y 698.098,Z 1136.974,A -85,B 0,C 180,E1 3489.429,E2 3489.429} C_VEL
LIN {X 0,Y 697.295,Z 1162.95,A -85,B 0,C 180,E1 3493.33,E2 3493.33} C_VEL
LIN {X 0,Y 696.828,Z 1182.48,A -85,B 0,C 180,E1 3497.189,E2 3497.189} C_VEL
LIN {X 0,Y 696.71,Z 1196.131,A -85,B 0,C 180,E1 3500.863,E2 3500.863} C_VEL
LIN {X 0,Y 696.597,Z 1204.797,A -85,B 0,C 180,E1 3504.397,E2 3504.397} C_VEL
LIN {X 0,Y 696.594,Z 1208.957,A -85,B 0,C 180,E1 3507.513,E2 3507.513} C_VEL
LIN {X 0,Y 696.73,Z 1209.669,A -85,B 0,C 180,E1 3511.242,E2 3511.242} C_VEL
LIN {X 0,Y 696.536,Z 1205.912,A -85,B 0,C 180,E1 3514.978,E2 3514.978} C_VEL
LIN {X 0,Y 696.562,Z 1197.334,A -85,B 0,C 180,E1 3518.734,E2 3518.734} C_VEL
LIN {X 0,Y 696.686,Z 1185.051,A -85,B 0,C 180,E1 3522.208,E2 3522.208} C_VEL
LIN {X 0,Y 697.082,Z 1167.227,A -85,B 0,C 180,E1 3525.905,E2 3525.905} C_VEL
LIN {X 0,Y 697.745,Z 1144.906,A -85,B 0,C 180,E1 3529.49,E2 3529.49} C_VEL
LIN {X 0,Y 698.719,Z 1116.141,A -85,B 0,C 180,E1 3533.141,E2 3533.141} C_VEL
LIN {X 0,Y 700.19,Z 1082.946,A -85,B 0,C 180,E1 3536.55,E2 3536.55} C_VEL
LIN {X 0,Y 702.055,Z 1043.513,A -85,B 0,C 180,E1 3539.798,E2 3539.798} C_VEL
LIN {X 0,Y 703.985,Z 1003.577,A -85,B 0,C 180,E1 3542.454,E2 3542.454} C_VEL
LIN {X 0,Y 706.092,Z 959.756,A -85,B 0,C 180,E1 3544.755,E2 3544.755} C_VEL
LIN {X 0,Y 707.909,Z 916.927,A -85,B 0,C 180,E1 3546.494,E2 3546.494} C_VEL
LIN {X 0,Y 709.301,Z 873.143,A -85,B 0,C 180,E1 3547.801,E2 3547.801} C_VEL
LIN {X 0,Y 710.321,Z 827.188,A -85,B 0,C 180,E1 3548.692,E2 3548.692} C_VEL
LIN {X 0,Y 710.082,Z 776.214,A -85,B 0,C 180,E1 3549.378,E2 3549.378} C_VEL
LIN {X 0,Y 696.183,Z 750.873,A -85,B 0,C 180,E1 3550.66,E2 3550.66} C_VEL
LIN {X 0,Y 696.099,Z 749.56,A -85,B 0,C 180,E1 3550.773,E2 3550.773} C_VEL
LIN {X 0,Y 696.17,Z 749.56,A -85,B 0,C 180,E1 3555.75,E2 3555.75} C_VEL
LIN {X 0,Y 696.131,Z 749.56,A -85,B 0,C 180,E1 3561.394,E2 3561.394} C_VEL
LIN {X 0,Y 696.049,Z 749.56,A -85,B 0,C 180,E1 3565.638,E2 3565.638} C_VEL
LIN {X 0,Y 696.102,Z 749.56,A -85,B 0,C 180,E1 3570.265,E2 3570.265} C_VEL
LIN {X 0,Y 696.121,Z 749.56,A -85,B 0,C 180,E1 3575.644,E2 3575.644} C_VEL
LIN {X 0,Y 696.164,Z 749.56,A -85,B 0,C 180,E1 3581.001,E2 3581.001} C_VEL
LIN {X 0,Y 696.348,Z 749.56,A -85,B 0,C 180,E1 3584.909,E2 3584.909} C_VEL
LIN {X 0,Y 696.377,Z 749.56,A -85,B 0,C 180,E1 3590.006,E2 3590.006} C_VEL
LIN {X 0,Y 696.613,Z 749.56,A -85,B 0,C 180,E1 3595.026,E2 3595.026} C_VEL
LIN {X 0,Y 696.494,Z 749.56,A -85,B 0,C 180,E1 3600.003,E2 3600.003} C_VEL
LIN {X 0,Y 696.428,Z 749.56,A -85,B 0,C 180,E1 3604.983,E2 3604.983} C_VEL
LIN {X 0,Y 696.452,Z 749.56,A -85,B 0,C 180,E1 3610,E2 3610} C_VEL
LIN {X 0,Y 696.175,Z 749.56,A -85,B 0,C 180,E1 3615.102,E2 3615.102} C_VEL
LIN {X 0,Y 696.123,Z 749.56,A -85,B 0,C 180,E1 3621.025,E2 3621.025} C_VEL
LIN {X 0,Y 696.057,Z 749.56,A -85,B 0,C 180,E1 3625.739,E2 3625.739} C_VEL
LIN {X 0,Y 696.091,Z 749.56,A -85,B 0,C 180,E1 3629.959,E2 3629.959} C_VEL
LIN {X 0,Y 696.049,Z 749.56,A -85,B 0,C 180,E1 3634.414,E2 3634.414} C_VEL
LIN {X 0,Y 696.143,Z 749.56,A -85,B 0,C 180,E1 3639.019,E2 3639.019} C_VEL
LIN {X 0,Y 696.255,Z 749.56,A -85,B 0,C 180,E1 3644.833,E2 3644.833} C_VEL
LIN {X 0,Y 707.884,Z 775.079,A -85,B 0,C 180,E1 3645.852,E2 3645.852} C_VEL
LIN {X 0,Y 707.039,Z 824.218,A -85,B 0,C 180,E1 3646.766,E2 3646.766} C_VEL
LIN {X 0,Y 705.644,Z 870.849,A -85,B 0,C 180,E1 3648.195,E2 3648.195} C_VEL
LIN {X 0,Y 703.874,Z 913.891,A -85,B 0,C 180,E1 3650.023,E2 3650.023} C_VEL
LIN {X 0,Y 702.079,Z 958.009,A -85,B 0,C 180,E1 3652.516,E2 3652.516} C_VEL
LIN {X 0,Y 700.352,Z 996.625,A -85,B 0,C 180,E1 3655.323,E2 3655.323} C_VEL
LIN {X 0,Y 699.05,Z 1029.141,A -85,B 0,C 180,E1 3658.271,E2 3658.271} C_VEL
LIN {X 0,Y 697.934,Z 1059.511,A -85,B 0,C 180,E1 3661.702,E2 3661.702} C_VEL
LIN {X 0,Y 697.18,Z 1084.415,A -85,B 0,C 180,E1 3665.315,E2 3665.315} C_VEL
LIN {X 0,Y 696.884,Z 1103.038,A -85,B 0,C 180,E1 3668.827,E2 3668.827} C_VEL
LIN {X 0,Y 696.601,Z 1116.382,A -85,B 0,C 180,E1 3672.321,E2 3672.321} C_VEL
LIN {X 0,Y 696.546,Z 1125.873,A -85,B 0,C 180,E1 3676.194,E2 3676.194} C_VEL
LIN {X 0,Y 696.489,Z 1129.75,A -85,B 0,C 180,E1 3680.005,E2 3680.005} C_VEL
LIN {X 0,Y 696.633,Z 1128.527,A -85,B 0,C 180,E1 3683.774,E2 3683.774} C_VEL
LIN {X 0,Y 696.615,Z 1122.139,A -85,B 0,C 180,E1 3687.514,E2 3687.514} C_VEL
LIN {X 0,Y 696.678,Z 1110.64,A -85,B 0,C 180,E1 3691.243,E2 3691.243} C_VEL
LIN {X 0,Y 696.976,Z 1095.223,A -85,B 0,C 180,E1 3694.683,E2 3694.683} C_VEL
LIN {X 0,Y 697.486,Z 1072.682,A -85,B 0,C 180,E1 3698.41,E2 3698.41} C_VEL
LIN {X 0,Y 698.328,Z 1047.126,A -85,B 0,C 180,E1 3701.705,E2 3701.705} C_VEL
LIN {X 0,Y 699.664,Z 1013.447,A -85,B 0,C 180,E1 3705.148,E2 3705.148} C_VEL
LIN {X 0,Y 701.324,Z 975.338,A -85,B 0,C 180,E1 3708.214,E2 3708.214} C_VEL
LIN {X 0,Y 703.12,Z 934.558,A -85,B 0,C 180,E1 3710.794,E2 3710.794} C_VEL
LIN {X 0,Y 704.88,Z 892.774,A -85,B 0,C 180,E1 3712.849,E2 3712.849} C_VEL
LIN {X 0,Y 706.439,Z 848.994,A -85,B 0,C 180,E1 3714.445,E2 3714.445} C_VEL
LIN {X 0,Y 707.581,Z 804.263,A -85,B 0,C 180,E1 3715.578,E2 3715.578} C_VEL
LIN {X 0,Y 707.438,Z 773.539,A -85,B 0,C 180,E1 3716.106,E2 3716.106} C_VEL
LIN {X 0,Y 696.301,Z 751.154,A -85,B 0,C 180,E1 3717.043,E2 3717.043} C_VEL
LIN {X 0,Y 696.121,Z 749.56,A -85,B 0,C 180,E1 3717.121,E2 3717.121} C_VEL
LIN {X 0,Y 696.141,Z 749.56,A -85,B 0,C 180,E1 3722.15,E2 3722.15} C_VEL
LIN {X 0,Y 696.125,Z 749.56,A -85,B 0,C 180,E1 3727.432,E2 3727.432} C_VEL
LIN {X 0,Y 696.204,Z 749.56,A -85,B 0,C 180,E1 3732.434,E2 3732.434} C_VEL
LIN {X 0,Y 695.998,Z 749.56,A -85,B 0,C 180,E1 3737.69,E2 3737.69} C_VEL
LIN {X 0,Y 696.075,Z 749.56,A -85,B 0,C 180,E1 3742.56,E2 3742.56} C_VEL
LIN {X 0,Y 696.011,Z 749.56,A -85,B 0,C 180,E1 3747.86,E2 3747.86} C_VEL
LIN {X 0,Y 696.099,Z 749.56,A -85,B 0,C 180,E1 3752.881,E2 3752.881} C_VEL
LIN {X 0,Y 696.038,Z 749.56,A -85,B 0,C 180,E1 3758.337,E2 3758.337} C_VEL
LIN {X 0,Y 695.994,Z 749.56,A -85,B 0,C 180,E1 3763.601,E2 3763.601} C_VEL
LIN {X 0,Y 696.402,Z 749.56,A -85,B 0,C 180,E1 3768.734,E2 3768.734} C_VEL
LIN {X 0,Y 696.543,Z 749.56,A -85,B 0,C 180,E1 3773.769,E2 3773.769} C_VEL
LIN {X 0,Y 696.445,Z 749.56,A -85,B 0,C 180,E1 3778.753,E2 3778.753} C_VEL
LIN {X 0,Y 696.446,Z 749.56,A -85,B 0,C 180,E1 3782.484,E2 3782.484} C_VEL
LIN {X 0,Y 696.434,Z 749.56,A -85,B 0,C 180,E1 3786.225,E2 3786.225} C_VEL
LIN {X 0,Y 696.335,Z 749.56,A -85,B 0,C 180,E1 3791.26,E2 3791.26} C_VEL
LIN {X 0,Y 696.413,Z 749.56,A -85,B 0,C 180,E1 3796.381,E2 3796.381} C_VEL
LIN {X 0,Y 696.428,Z 749.56,A -85,B 0,C 180,E1 3797.225,E2 3797.225} C_VEL
LIN {X 0,Y 693.915,Z 749.56,A -85,B 0,C 180,E1 3798.284,E2 3798.284} C_VEL
LIN {X 0,Y 688.49,Z 749.56,A -85,B 0,C 180,E1 3799.864,E2 3799.864} C_VEL
LIN {X 0,Y 688.4,Z 749.56,A -85,B 0,C 180,E1 3800.047,E2 3800.047} C_VEL
LIN {X 0,Y 688.373,Z 749.56,A -85,B 0,C 180,E1 3804.648,E2 3804.648} C_VEL
LIN {X 0,Y 688.312,Z 749.56,A -85,B 0,C 180,E1 3808.878,E2 3808.878} C_VEL
LIN {X 0,Y 688.263,Z 749.56,A -85,B 0,C 180,E1 3813.454,E2 3813.454} C_VEL
LIN {X 0,Y 688.192,Z 749.56,A -85,B 0,C 180,E1 3817.936,E2 3817.936} C_VEL
LIN {X 0,Y 688.319,Z 749.56,A -85,B 0,C 180,E1 3823.574,E2 3823.574} C_VEL
LIN {X 0,Y 688.232,Z 749.803,A -85,B 0,C 180,E1 3828.754,E2 3828.754} C_VEL
LIN {X 0,Y 693.072,Z 759.853,A -85,B 0,C 180,E1 3829.239,E2 3829.239} C_VEL
LIN {X 0,Y 704.505,Z 780.611,A -85,B 0,C 180,E1 3830.305,E2 3830.305} C_VEL
LIN {X 0,Y 703.825,Z 848.559,A -85,B 0,C 180,E1 3831.272,E2 3831.272} C_VEL
LIN {X 0,Y 702.25,Z 892.011,A -85,B 0,C 180,E1 3832.301,E2 3832.301} C_VEL
LIN {X 0,Y 700.37,Z 938.494,A -85,B 0,C 180,E1 3833.93,E2 3833.93} C_VEL
LIN {X 0,Y 698.062,Z 985.633,A -85,B 0,C 180,E1 3836.163,E2 3836.163} C_VEL
LIN {X 0,Y 695.772,Z 1027.052,A -85,B 0,C 180,E1 3838.687,E2 3838.687} C_VEL
LIN {X 0,Y 693.591,Z 1067.81,A -85,B 0,C 180,E1 3841.797,E2 3841.797} C_VEL
LIN {X 0,Y 691.766,Z 1103.226,A -85,B 0,C 180,E1 3845.167,E2 3845.167} C_VEL
LIN {X 0,Y 690.495,Z 1134.083,A -85,B 0,C 180,E1 3848.793,E2 3848.793} C_VEL
LIN {X 0,Y 689.574,Z 1161.403,A -85,B 0,C 180,E1 3852.877,E2 3852.877} C_VEL
LIN {X 0,Y 689.064,Z 1180.994,A -85,B 0,C 180,E1 3856.687,E2 3856.687} C_VEL
LIN {X 0,Y 688.828,Z 1196.279,A -85,B 0,C 180,E1 3860.808,E2 3860.808} C_VEL
LIN {X 0,Y 688.732,Z 1204.797,A -85,B 0,C 180,E1 3864.333,E2 3864.333} C_VEL
LIN {X 0,Y 688.691,Z 1208.954,A -85,B 0,C 180,E1 3867.484,E2 3867.484} C_VEL
LIN {X 0,Y 688.848,Z 1209.669,A -85,B 0,C 180,E1 3871.256,E2 3871.256} C_VEL
LIN {X 0,Y 688.635,Z 1205.912,A -85,B 0,C 180,E1 3875.035,E2 3875.035} C_VEL
LIN {X 0,Y 688.686,Z 1197.333,A -85,B 0,C 180,E1 3878.835,E2 3878.835} C_VEL
LIN {X 0,Y 688.836,Z 1185.109,A -85,B 0,C 180,E1 3882.336,E2 3882.336} C_VEL
LIN {X 0,Y 689.276,Z 1166.647,A -85,B 0,C 180,E1 3886.198,E2 3886.198} C_VEL
LIN {X 0,Y 690.047,Z 1144.534,A -85,B 0,C 180,E1 3889.773,E2 3889.773} C_VEL
LIN {X 0,Y 691.217,Z 1115.022,A -85,B 0,C 180,E1 3893.536,E2 3893.536} C_VEL
LIN {X 0,Y 692.851,Z 1081.981,A -85,B 0,C 180,E1 3896.943,E2 3896.943} C_VEL
LIN {X 0,Y 695.021,Z 1041.086,A -85,B 0,C 180,E1 3900.321,E2 3900.321} C_VEL
LIN {X 0,Y 697.229,Z 999.76,A -85,B 0,C 180,E1 3903.041,E2 3903.041} C_VEL
LIN {X 0,Y 699.674,Z 954.563,A -85,B 0,C 180,E1 3905.379,E2 3905.379} C_VEL
LIN {X 0,Y 701.622,Z 912.24,A -85,B 0,C 180,E1 3907.047,E2 3907.047} C_VEL
LIN {X 0,Y 703.088,Z 869.821,A -85,B 0,C 180,E1 3908.281,E2 3908.281} C_VEL
LIN {X 0,Y 704.209,Z 823.315,A -85,B 0,C 180,E1 3909.15,E2 3909.15} C_VEL
LIN {X 0,Y 703.875,Z 779.385,A -85,B 0,C 180,E1 3909.753,E2 3909.753} C_VEL
LIN {X 0,Y 688.447,Z 751.18,A -85,B 0,C 180,E1 3911.212,E2 3911.212} C_VEL
LIN {X 0,Y 688.28,Z 749.56,A -85,B 0,C 180,E1 3911.301,E2 3911.301} C_VEL
LIN {X 0,Y 688.173,Z 749.56,A -85,B 0,C 180,E1 3916.437,E2 3916.437} C_VEL
LIN {X 0,Y 688.196,Z 749.56,A -85,B 0,C 180,E1 3922.229,E2 3922.229} C_VEL
LIN {X 0,Y 688.099,Z 749.56,A -85,B 0,C 180,E1 3926.703,E2 3926.703} C_VEL
LIN {X 0,Y 688.185,Z 749.56,A -85,B 0,C 180,E1 3931.44,E2 3931.44} C_VEL
LIN {X 0,Y 688.201,Z 749.56,A -85,B 0,C 180,E1 3936.722,E2 3936.722} C_VEL
LIN {X 0,Y 688.346,Z 749.56,A -85,B 0,C 180,E1 3942.104,E2 3942.104} C_VEL
LIN {X 0,Y 688.489,Z 749.56,A -85,B 0,C 180,E1 3947.324,E2 3947.324} C_VEL
LIN {X 0,Y 688.508,Z 749.56,A -85,B 0,C 180,E1 3952.436,E2 3952.436} C_VEL
LIN {X 0,Y 688.597,Z 749.56,A -85,B 0,C 180,E1 3956.229,E2 3956.229} C_VEL
LIN {X 0,Y 688.618,Z 749.56,A -85,B 0,C 180,E1 3960.003,E2 3960.003} C_VEL
LIN {X 0,Y 688.526,Z 749.56,A -85,B 0,C 180,E1 3965.04,E2 3965.04} C_VEL
LIN {X 0,Y 688.543,Z 749.56,A -85,B 0,C 180,E1 3970.116,E2 3970.116} C_VEL
LIN {X 0,Y 688.243,Z 749.56,A -85,B 0,C 180,E1 3975.28,E2 3975.28} C_VEL
LIN {X 0,Y 688.234,Z 749.56,A -85,B 0,C 180,E1 3980.571,E2 3980.571} C_VEL
LIN {X 0,Y 688.146,Z 749.56,A -85,B 0,C 180,E1 3986.057,E2 3986.057} C_VEL
LIN {X 0,Y 688.129,Z 749.56,A -85,B 0,C 180,E1 3991.082,E2 3991.082} C_VEL
LIN {X 0,Y 688.124,Z 749.56,A -85,B 0,C 180,E1 3996.37,E2 3996.37} C_VEL
LIN {X 0,Y 688.07,Z 749.56,A -85,B 0,C 180,E1 4001.695,E2 4001.695} C_VEL
LIN {X 0,Y 688.243,Z 749.56,A -85,B 0,C 180,E1 4004.356,E2 4004.356} C_VEL
LIN {X 0,Y 694.392,Z 762.907,A -85,B 0,C 180,E1 4004.9,E2 4004.9} C_VEL
LIN {X 0,Y 701.431,Z 778.449,A -85,B 0,C 180,E1 4005.53,E2 4005.53} C_VEL
LIN {X 0,Y 700.431,Z 824.903,A -85,B 0,C 180,E1 4006.417,E2 4006.417} C_VEL
LIN {X 0,Y 698.884,Z 871.228,A -85,B 0,C 180,E1 4007.852,E2 4007.852} C_VEL
LIN {X 0,Y 696.901,Z 914.654,A -85,B 0,C 180,E1 4009.72,E2 4009.72} C_VEL
LIN {X 0,Y 694.89,Z 958.526,A -85,B 0,C 180,E1 4012.228,E2 4012.228} C_VEL
LIN {X 0,Y 692.864,Z 998.598,A -85,B 0,C 180,E1 4015.19,E2 4015.19} C_VEL
LIN {X 0,Y 691.294,Z 1032.516,A -85,B 0,C 180,E1 4018.358,E2 4018.358} C_VEL
LIN {X 0,Y 690.136,Z 1061.477,A -85,B 0,C 180,E1 4021.739,E2 4021.739} C_VEL
LIN {X 0,Y 689.328,Z 1085.935,A -85,B 0,C 180,E1 4025.386,E2 4025.386} C_VEL
LIN {X 0,Y 688.968,Z 1104.422,A -85,B 0,C 180,E1 4029.015,E2 4029.015} C_VEL
LIN {X 0,Y 688.686,Z 1117.369,A -85,B 0,C 180,E1 4032.546,E2 4032.546} C_VEL
LIN {X 0,Y 688.655,Z 1125.67,A -85,B 0,C 180,E1 4036.033,E2 4036.033} C_VEL
LIN {X 0,Y 688.583,Z 1129.722,A -85,B 0,C 180,E1 4039.889,E2 4039.889} C_VEL
LIN {X 0,Y 688.725,Z 1128.612,A -85,B 0,C 180,E1 4043.702,E2 4043.702} C_VEL
LIN {X 0,Y 688.722,Z 1122.396,A -85,B 0,C 180,E1 4047.486,E2 4047.486} C_VEL
LIN {X 0,Y 688.806,Z 1111.018,A -85,B 0,C 180,E1 4051.258,E2 4051.258} C_VEL
LIN {X 0,Y 689.119,Z 1095.395,A -85,B 0,C 180,E1 4054.81,E2 4054.81} C_VEL
LIN {X 0,Y 689.703,Z 1073.402,A -85,B 0,C 180,E1 4058.505,E2 4058.505} C_VEL
LIN {X 0,Y 690.628,Z 1048.077,A -85,B 0,C 180,E1 4061.838,E2 4061.838} C_VEL
LIN {X 0,Y 692.123,Z 1014.578,A -85,B 0,C 180,E1 4065.323,E2 4065.323} C_VEL
LIN {X 0,Y 694.012,Z 976.236,A -85,B 0,C 180,E1 4068.457,E2 4068.457} C_VEL
LIN {X 0,Y 695.914,Z 937.424,A -85,B 0,C 180,E1 4070.965,E2 4070.965} C_VEL
LIN {X 0,Y 697.943,Z 894.976,A -85,B 0,C 180,E1 4073.106,E2 4073.106} C_VEL
LIN {X 0,Y 699.699,Z 850.869,A -85,B 0,C 180,E1 4074.749,E2 4074.749} C_VEL
LIN {X 0,Y 701.04,Z 805.125,A -85,B 0,C 180,E1 4075.932,E2 4075.932} C_VEL
LIN {X 0,Y 700.987,Z 776.491,A -85,B 0,C 180,E1 4076.435,E2 4076.435} C_VEL
LIN {X 0,Y 688.326,Z 750.937,A -85,B 0,C 180,E1 4077.531,E2 4077.531} C_VEL
LIN {X 0,Y 688.201,Z 749.56,A -85,B 0,C 180,E1 4077.598,E2 4077.598} C_VEL
LIN {X 0,Y 688.219,Z 749.56,A -85,B 0,C 180,E1 4081.802,E2 4081.802} C_VEL
LIN {X 0,Y 688.18,Z 749.56,A -85,B 0,C 180,E1 4086.362,E2 4086.362} C_VEL
LIN {X 0,Y 688.171,Z 749.56,A -85,B 0,C 180,E1 4091.697,E2 4091.697} C_VEL
LIN {X 0,Y 688.129,Z 749.56,A -85,B 0,C 180,E1 4096.443,E2 4096.443} C_VEL
LIN {X 0,Y 688.176,Z 749.56,A -85,B 0,C 180,E1 4102.234,E2 4102.234} C_VEL
LIN {X 0,Y 688.087,Z 749.56,A -85,B 0,C 180,E1 4106.694,E2 4106.694} C_VEL
LIN {X 0,Y 688.16,Z 749.56,A -85,B 0,C 180,E1 4111.446,E2 4111.446} C_VEL
LIN {X 0,Y 688.092,Z 749.56,A -85,B 0,C 180,E1 4115.334,E2 4115.334} C_VEL
LIN {X 0,Y 688.175,Z 749.56,A -85,B 0,C 180,E1 4120.774,E2 4120.774} C_VEL
LIN {X 0,Y 688.278,Z 749.56,A -85,B 0,C 180,E1 4126.021,E2 4126.021} C_VEL
LIN {X 0,Y 688.475,Z 749.56,A -85,B 0,C 180,E1 4131.158,E2 4131.158} C_VEL
LIN {X 0,Y 688.613,Z 749.56,A -85,B 0,C 180,E1 4136.222,E2 4136.222} C_VEL
LIN {X 0,Y 688.8,Z 749.56,A -85,B 0,C 180,E1 4141.254,E2 4141.254} C_VEL
LIN {X 0,Y 688.524,Z 749.56,A -85,B 0,C 180,E1 4146.297,E2 4146.297} C_VEL
LIN {X 0,Y 688.443,Z 749.56,A -85,B 0,C 180,E1 4151.39,E2 4151.39} C_VEL
LIN {X 0,Y 688.505,Z 749.56,A -85,B 0,C 180,E1 4156.575,E2 4156.575} C_VEL
